Yaskawa INFORM job: OK_R2_O57-69(1)(90,0)_OK_HARDOX.JBI

/JOB
//NAME OK_R2_O57-69(1)(90,0)_OK_HARDOX
///FOLDERNAME X4
//POS
///NPOS 554,554,554,23,0,0
///TOOL 0
///POSTYPE PULSE
///PULSE
C00000=-107863,126513,61876,4074,92941,-4149
C00001=-107635,120046,52933,4022,95106,-4012
C00002=-107385,124787,62548,3925,91623,-4047
C00003=-107289,126429,66937,3891,89767,-4074
C00004=-107289,125685,67059,3890,89310,-4088
C00005=-107289,126429,66937,3891,89767,-4074
C00006=-107447,131976,74605,3936,87910,-4183
C00007=-107368,129085,70604,3913,88881,-4126
C00008=-107503,121805,59343,3962,92067,-4069
C00009=-107756,117289,50059,4061,95463,-4036
C00010=-108153,112100,52912,9904,92668,-10418
C00011=-107537,116907,62411,9707,89272,-10490
C00012=-107296,118643,67053,9639,87306,-10566
C00013=-107296,118210,67408,9641,86871,-10599
C00014=-107296,118643,67053,9639,87306,-10566
C00015=-106873,123308,73383,9530,85780,-10546
C00016=-107051,120523,69599,9574,86686,-10534
C00017=-107734,114067,59645,9761,89532,-10533
C00018=-108357,109439,50420,9963,92855,-10467
C00019=-111395,93808,29792,10909,97789,-10982
C00020=-122185,34205,35653,27729,49230,-19016
C00021=-120981,41909,45488,27980,46968,-19127
C00022=-117396,66636,64308,14609,59928,-14205
C00023=-117396,67398,66227,14722,59162,-14310
C00024=-117396,66924,65038,14651,59635,-14244
C00025=-117026,69424,68003,14605,59045,-14176
C00026=-117396,66924,65038,14651,59635,-14244
C00027=-121567,39659,44448,28509,46708,-19512
C00028=-122801,32028,34766,28268,48928,-19417
C00029=-122836,-30084,-33960,23424,71784,-41222
C00030=-108542,-18181,-29050,8736,76414,-35911
C00031=-108679,-18112,-25517,8852,74315,-36109
C00032=-108679,-17878,-23614,8896,73277,-36184
C00033=-108679,-18015,-24674,8871,73853,-36141
C00034=-101227,-12151,-22997,-5627,79968,-34149
C00035=-100809,-11793,-21323,-5732,79157,-33969
C00036=-99890,-11248,-20900,-5932,79243,-33658
C00037=-100809,-11793,-21323,-5732,79157,-33969
C00038=-119599,-28607,-38623,18108,79564,-38965
C00039=-143809,-13353,-27562,-4151,73883,-14363
C00040=-142866,3813,-3489,-4615,67955,-13814
C00041=-142866,4258,-993,-4658,66653,-13764
C00042=-142866,4067,-2013,-4640,67181,-13786
C00043=-143013,7668,1106,-4588,67106,-13835
C00044=-142866,4067,-2013,-4640,67181,-13786
C00045=-131729,19399,12333,-22118,77640,8494
C00046=-132684,19784,12695,-21959,77361,8191
C00047=-131729,18326,5882,-21907,80820,7904
C00048=-118180,-25123,-37779,-23861,88752,11312
C00049=-84402,-63677,-67114,-22586,99939,48241
C00050=-125926,-77250,-66316,-21080,81833,36437
C00051=-126284,-594,-20029,-15604,88354,35723
C00052=-126284,-509,-12976,-15645,84209,36248
C00053=-124802,3877,-7879,-15893,83645,36839
C00054=-124802,4020,-6552,-15911,82926,36931
C00055=-124802,3943,-7243,-15902,83298,36884
C00056=-123270,3785,-7378,-16131,83600,37383
C00057=-123399,3884,-6575,-16123,83149,37397
C00058=-123813,3922,-6544,-16060,83068,37263
C00059=-123399,3797,-7355,-16113,83568,37342
C00060=-129363,-46213,-49135,-15183,82438,35396
C00061=-131818,-93939,-91511,-4308,83147,7603
C00062=-129147,-104974,-80844,32439,31226,-48978
C00063=-125584,-72667,-62488,33742,33102,-67368
C00064=-122739,-67050,-57509,31022,31859,-65945
C00065=-121864,-64027,-53896,30654,30960,-65755
C00066=-121864,-63651,-52586,31182,30432,-66030
C00067=-121864,-64027,-53896,30654,30960,-65755
C00068=-121821,-59098,-51320,29827,31769,-65322
C00069=-121798,-56590,-49965,29444,32160,-65121
C00070=-121821,-59098,-51320,29827,31769,-65322
C00071=-130221,-55648,-47387,49393,39382,-72629
C00072=-128533,-55969,-47565,48393,38431,-72058
C00073=-122326,-63724,-54491,30711,31580,-65784
C00074=-123406,-65952,-56523,31749,32071,-66325
C00075=-126254,-71501,-61496,34397,33361,-67713
C00076=-120687,-90156,-48971,65843,10407,33929
C00077=-163424,-29173,-12092,69684,68620,47205
C00078=-167450,-15662,-2475,69350,71709,47134
C00079=-157670,-380,9649,68931,65290,48661
C00080=-176833,-62202,-56111,67907,81183,43629
C00081=-171503,-69579,-59831,67744,77015,43718
C00082=-167720,-72113,-59544,67781,73885,43604
C00083=-167720,-71727,-58313,67922,73661,43360
C00084=-167720,-72113,-59544,67781,73885,43604
C00085=-166558,-71597,-59299,67661,73156,43817
C00086=-165333,-70928,-58979,67520,72398,44056
C00087=-166558,-71597,-59299,67661,73156,43817
C00088=-171811,-70314,-60189,67797,77159,43607
C00089=-177694,-60868,-55413,67941,81861,43620
C00090=-178740,-64487,-57291,68086,82281,43176
C00091=-194893,-69888,-59984,68507,92693,40544
C00092=-214988,-85940,-67216,66402,104593,36100
C00093=-106040,-96827,-71490,56175,31560,53564
C00094=-84767,-92802,-92316,-2687,45777,78237
C00095=-91047,27807,-31300,-12206,82587,77963
C00096=-102219,10733,-36282,-6756,75834,75159
C00097=-102220,10108,-35615,-6792,75115,75199
C00098=-102220,9478,-34889,-6816,74349,75240
C00099=-102220,9734,-35191,-6806,74664,75222
C00100=-100300,10893,-34158,-7793,74779,75816
C00101=-100300,10587,-33794,-7807,74401,75842
C00102=-101147,10060,-34263,-7371,74347,75579
C00103=-101076,10802,-35034,-7381,75201,75550
C00104=-95480,80551,28809,-25074,106745,88551
C00105=-95760,77540,27472,-24942,106007,88613
C00106=-95760,76990,28122,-24849,105386,88749
C00107=-95760,77103,27982,-24868,105516,88720
C00108=-96959,80585,32244,-24647,104424,88528
C00109=-96959,80447,32426,-24624,104257,88565
C00110=-96409,78816,30426,-24722,104765,88651
C00111=-100062,100483,54273,-17494,109954,86476
C00112=-106835,71636,17530,-18824,115982,83026
C00113=-106612,70519,18025,-18669,115194,83244
C00114=-106612,70167,18360,-18604,114826,83306
C00115=-106612,70294,18237,-18628,114960,83283
C00116=-107711,74369,23131,-18489,113861,83072
C00117=-107711,74237,23265,-18465,113717,83098
C00118=-107290,72601,21292,-18521,114156,83175
C00119=-107383,75666,22241,-18686,115079,82983
C00120=-103109,12889,-33455,-26802,75758,89629
C00121=-108969,18301,-24187,-24197,71491,88552
C00122=-108969,17786,-23402,-24296,70807,88698
C00123=-108969,17914,-23607,-24271,70984,88661
C00124=-107778,14157,-27071,-24854,71490,88973
C00125=-107778,13979,-26794,-24889,71252,89025
C00126=-108147,15245,-25637,-24709,71092,88927
C00127=-108126,15683,-27040,-24578,72092,88718
C00128=-100567,37939,-6230,-27391,72804,90359
C00129=-100865,37186,-5596,-27353,72020,90442
C00130=-100865,36842,-5001,-27431,71534,90560
C00131=-100865,36955,-5200,-27406,71694,90520
C00132=-99747,33295,-8939,-27886,72410,90754
C00133=-99747,33126,-8648,-27924,72173,90813
C00134=-100160,34398,-7357,-27744,71921,90725
C00135=-100129,35026,-9173,-27563,73215,90418
C00136=-110911,33745,-10798,1686,65996,79969
C00137=-110596,33512,-9684,1507,65185,80063
C00138=-110596,33168,-9124,1512,64663,80058
C00139=-110596,33307,-9355,1509,64876,80061
C00140=-109674,30137,-12540,942,65194,80377
C00141=-109674,29950,-12234,942,64908,80377
C00142=-110141,31373,-10814,1228,64772,80217
C00143=-110010,31979,-12214,1138,65943,80273
C00144=-98269,67962,25517,-6197,61564,84446
C00145=-97899,69655,29924,-6541,59762,84684
C00146=-97899,69423,30622,-6575,59215,84716
C00147=-97899,69536,30274,-6557,59484,84700
C00148=-96720,65812,25908,-7249,60348,85083
C00149=-96720,65654,26340,-7274,60006,85106
C00150=-97107,66951,27854,-7050,59711,84981
C00151=-96963,66930,26864,-7100,60316,84996
C00152=-95444,-1255,-51083,-7343,73273,84703
C00153=-87441,-44243,-81586,-12090,70841,87391
C00154=-204042,-120915,-85873,62426,87530,23210
C00155=-200540,-66438,-67217,63628,100285,-15829
C00156=-127293,-88890,-117674,21964,112183,-47373
C00157=-127884,-113870,-117586,20406,100261,-49782
C00158=-126455,-94233,-83658,19548,96625,-49926
C00159=-122769,-95152,-80887,19686,93685,-49072
C00160=-121257,-92855,-76623,19731,91957,-48808
C00161=-121256,-92184,-75240,19721,91480,-48885
C00162=-121257,-92855,-76623,19731,91957,-48808
C00163=-119709,-92847,-76620,19813,91585,-48312
C00164=-118447,-92805,-76604,19874,91287,-47906
C00165=-121134,-93057,-78029,19757,92646,-48652
C00166=-122616,-92853,-79205,19699,93786,-49000
C00167=-126246,-91944,-81970,19569,96706,-49837
C00168=-116739,-91029,-87152,-11175,94833,69838
C00169=-118638,-93558,-84500,-11112,91693,69464
C00170=-121559,-94813,-81066,-11067,88585,68734
C00171=-121559,-94454,-79960,-11067,88097,68778
C00172=-121559,-94813,-81066,-11067,88585,68734
C00173=-121580,-97932,-82261,-11067,87731,68801
C00174=-121559,-94813,-81066,-11067,88585,68734
C00175=-124478,-94674,-81011,-11026,88221,67759
C00176=-121559,-94813,-81066,-11067,88585,68734
C00177=-121199,-93273,-83309,-11082,90766,68663
C00178=-119237,-90980,-86060,-11143,93854,69064
C00179=-119262,-91078,-98551,-11400,101347,68370
C00180=-119262,-88450,-105465,-11733,106843,67839
C00181=-123634,-129086,-124562,18007,62786,-21453
C00182=-124713,-112307,-109989,18584,62695,-21889
C00183=-121750,-102661,-104576,16897,63614,-20597
C00184=-120661,-96847,-100545,16291,63882,-20142
C00185=-120661,-96945,-99213,16408,63045,-20264
C00186=-120661,-96847,-100545,16291,63882,-20142
C00187=-119434,-96825,-100537,15680,63651,-19709
C00188=-118199,-96764,-100511,15059,63439,-19270
C00189=-119434,-96825,-100537,15680,63651,-19709
C00190=-120468,-95018,-99831,16130,64325,-20004
C00191=-120473,-92385,-98782,16042,65005,-19908
C00192=-120468,-95018,-99831,16130,64325,-20004
C00193=-121400,-102567,-103315,16828,62845,-20579
C00194=-124338,-112119,-108698,18515,61948,-21869
C00195=-115152,-110094,-108973,-21966,66789,27187
C00196=-118701,-101887,-103909,-20282,66922,25804
C00197=-120033,-96498,-99821,-19662,66842,25314
C00198=-120033,-96571,-98630,-19770,66116,25442
C00199=-120033,-96498,-99821,-19662,66842,25314
C00200=-121038,-96503,-99823,-19217,66607,24975
C00201=-122863,-96447,-99800,-18396,66209,24352
C00202=-121038,-96503,-99823,-19217,66607,24975
C00203=-121031,-93073,-98698,-19079,67622,24806
C00204=-121028,-91162,-97925,-19016,68103,24728
C00205=-121031,-93073,-98698,-19079,67622,24806
C00206=-119849,-101075,-102503,-19842,66224,25492
C00207=-116381,-109262,-107580,-21511,66068,26853
C00208=-114174,-113759,-109466,-25218,61256,29915
C00209=-117999,-105066,-104585,-23039,61495,28291
C00210=-119436,-99712,-100384,-22286,61259,27759
C00211=-119436,-99710,-99356,-22420,60673,27881
C00212=-119436,-99712,-100384,-22286,61259,27759
C00213=-121229,-99730,-100389,-21374,60785,27131
C00214=-123455,-99637,-100354,-20211,60254,26337
C00215=-121229,-99730,-100389,-21374,60785,27131
C00216=-121193,-87849,-97584,-20616,64895,26352
C00217=-121184,-85182,-96456,-20515,65531,26236
C00218=-121193,-87849,-97584,-20616,64895,26352
C00219=-119818,-94456,-100985,-21520,64018,27049
C00220=-116346,-102514,-105912,-23431,63914,28430
C00221=-120616,-96535,-104175,-23887,64719,45568
C00222=-120616,-96992,-102054,-24182,63306,45881
C00223=-136549,-91664,-102215,-2850,64532,40154
C00224=-118869,-97062,-101163,-25162,63282,46587
C00225=-120614,-98220,-102778,-24220,63138,45920
C00226=-133771,-94843,-111628,-11760,91195,37379
C00227=-135495,-95953,-105009,-10406,87462,38794
C00228=-135817,-95923,-103691,-10152,86855,39072
C00229=-120616,-96793,-103087,-23408,87451,42960
C00230=-120617,-96070,-105685,-23410,89266,42604
C00231=-120635,-118119,-124325,-17957,114364,37370
C00232=-107148,-122068,-106720,-37591,45003,56343
C00233=-107143,-118125,-97071,-40168,41922,57944
C00234=-107140,-117153,-94914,-40772,41285,58308
C00235=-108761,-111076,-92035,-38763,41593,57087
C00236=-105115,-116142,-93852,-42098,42144,59139
C00237=-107012,-118507,-95796,-40965,41228,58425
C00238=-106625,-124982,-112623,-27698,77800,49761
C00239=-108670,-124346,-112001,-25564,83023,48254
C00240=-122914,-112386,-108022,-9565,118901,48106
C00241=-107149,-124464,-114807,-14035,115464,42498
C00242=-107153,-124980,-118069,-14274,117155,42276
C00243=-120683,-72727,-118704,-1403,106780,1205
C00244=-120616,-97084,-101761,23685,56760,-46645
C00245=-120615,-97341,-97713,24403,54354,-47226
C00246=-120615,-97245,-95574,24781,53197,-47519
C00247=-113473,-96585,-93861,15515,48754,-41599
C00248=-120613,-98403,-96349,24817,53089,-47545
C00249=-122362,-97151,-94697,25998,53280,-48291
C00250=-118726,-95773,-106258,22948,89010,-41713
C00251=-118527,-107245,-109313,22939,85243,-42364
C00252=-120617,-95328,-107797,23350,90604,-42068
C00253=-120618,-93989,-110172,23402,92584,-41681
C00254=-120619,-87370,-116055,23793,99045,-40394
C00255=-120619,-87370,-116055,23793,99045,-40394
C00256=-120618,-86394,-114990,-8935,74593,-77376
C00257=-120618,-89943,-112390,-9089,71210,-77123
C00258=-120618,-91094,-111253,-9157,69935,-77026
C00259=-120921,-87010,-110025,-8929,71231,-77225
C00260=-120616,-91696,-112687,-9127,70502,-77069
C00261=-120617,-91433,-110915,-9280,69085,-76949
C00262=-120617,-91707,-110620,-9342,68290,-76888
C00263=-120617,-92092,-110153,-9289,66860,-76810
C00264=-120617,-92703,-109346,-8604,64312,-76688
C00265=-120617,-93084,-108807,-7222,62458,-76641
C00266=-120617,-93193,-108666,-5837,61715,-76664
C00267=-120618,-90875,-111661,-5103,64613,-76670
C00268=-120618,-90809,-111742,-4197,64653,-76687
C00269=-120618,-90545,-112027,-2634,65244,-76730
C00270=-120618,-90001,-112556,-1051,66686,-76779
C00271=-120618,-89211,-113241,130,68806,-76818
C00272=-120618,-88484,-113805,667,70701,-76840
C00273=-120618,-87123,-114601,725,72803,-76709
C00274=-120619,-86169,-115177,666,75079,-76754
C00275=-120619,-85009,-115798,-44,77805,-76866
C00276=-120619,-84186,-116189,-1368,79788,-77043
C00277=-120619,-83945,-116287,-2643,80551,-77203
C00278=-118270,-87908,-113898,-4548,77310,-76315
C00279=-117006,-87882,-113777,-5977,77383,-75992
C00280=-115001,-87936,-113393,-8376,77055,-75464
C00281=-113157,-88199,-112730,-10795,75966,-74930
C00282=-112003,-88721,-111920,-12625,74164,-74513
C00283=-111959,-89151,-111512,-13141,72976,-74431
C00284=-114352,-90005,-111461,-12180,71784,-75105
C00285=-117604,-90791,-111341,-10710,70486,-76060
C00286=-117404,-89600,-112462,-10735,71791,-76111
C00287=-116906,-85938,-115017,-10812,75246,-76259
C00288=-120614,-97623,-100799,-20300,88883,51757
C00289=-120614,-96302,-87355,-20440,81742,52958
C00290=-120613,-95405,-83784,-20521,80111,53236
C00291=-127344,-108772,-84900,-17713,65232,40253
C00292=-119108,-93712,-82042,-20736,80300,53753
C00293=-120703,-96440,-84059,-20528,79748,53266
C00294=-121654,-94959,-82200,-16195,85067,56749
C00295=-121447,-94482,-79045,-16244,83477,57034
C00296=-120534,-97306,-80078,-13287,88870,68293
C00297=-120613,-95181,-82964,-13310,91650,67966
C00298=-120614,-96223,-86939,-13345,93512,67766
C00299=-120615,-97634,-95801,-13498,98116,67263
C00300=-121294,-114205,-91205,24827,58618,-34956
C00301=-120612,-94063,-79189,30374,49118,-27390
C00302=-120612,-92317,-74276,31337,47279,-28045
C00303=-120611,-91635,-72532,31685,46659,-28276
C00304=-117825,-85297,-69483,27706,45876,-25590
C00305=-120609,-92794,-73597,31655,46709,-28256
C00306=-122365,-91337,-71823,32796,47086,-29053
C00307=-115287,-110447,-90354,20374,67075,-37718
C00308=-116232,-100454,-77072,21254,66209,-40580
C00309=-116013,-94136,-76050,20295,81458,-56297
C00310=-120612,-93792,-78416,23522,88402,-60481
C00311=-120613,-94966,-82014,23532,89885,-60189
C00312=-192979,-49879,-84133,31949,90821,-59300
C00313=-226136,-49296,-77583,43048,96139,-60221
C00314=-194231,-43574,-37464,64429,96533,35524
C00315=-168190,-921,2356,69742,86936,65420
C00316=-167171,-9679,-4727,69794,80481,66551
C00317=-161668,-12899,-4972,71887,72051,48991
C00318=-157343,-12771,-6150,68681,68498,39910
C00319=-156881,-17849,-10944,69825,79076,66625
C00320=-156054,-17027,-11609,69675,78824,67093
C00321=-157320,-12846,-6207,68680,68481,39912
C00322=-155303,-14498,-7398,68413,65801,40416
C00323=-150761,-18705,-10675,67104,57790,42164
C00324=-154138,4950,8277,69166,76187,38481
C00325=-154445,-11009,-7055,66235,75211,55885
C00326=-154064,-10379,-10377,61252,81435,65690
C00327=-159305,-13086,-7363,68622,70046,39902
C00328=-160610,-11568,-6196,68690,70948,39749
C00329=-179726,-19719,-12316,69264,83687,37039
C00330=-180202,-65513,-36112,70171,79517,38597
C00331=-171321,-47804,-23743,70196,73038,45095
C00332=-120855,-117042,-83065,287,50429,-281
C00333=-120852,-56541,-79529,233,79340,-219
C00334=-120696,51333,26745,175,69370,-180
C00335=-120686,107911,74673,172,68949,-177
C00336=-120685,95088,60632,169,71000,-174
C00337=-122318,97205,64688,817,69601,-751
C00338=-120685,108202,77433,173,67399,-179
C00339=-120704,104217,73450,180,67803,-185
C00340=-122286,97202,64700,804,69591,-740
C00341=-121454,98107,65862,475,69334,-448
C00342=-120585,97922,65623,2034,69446,-1841
C00343=-122017,99369,67601,7878,69886,-7136
C00344=-124401,105713,75936,15606,71119,-14640
C00345=-128119,115493,91326,26372,70058,-18277
C00346=-128088,115464,91288,26362,70055,-18265
C00347=-119886,111402,95174,38234,57086,-30403
C00348=-120666,108818,81293,29360,75518,-26461
C00349=-140740,108253,75800,14319,69459,-12393
C00350=-141155,96820,62941,14306,71509,-12294
C00351=-143909,115216,86261,19079,74712,-18279
C00352=-140740,108512,78347,14450,68068,-12565
C00353=-141173,105757,75971,14609,68190,-12710
C00354=-142377,104065,71962,18453,77277,-17320
C00355=-143915,117471,89727,22794,77825,-23537
C00356=-139477,109798,84410,35996,86879,-36501
C00357=-140751,108928,81956,36051,87607,-36108
C00358=-140752,108346,78971,36051,88864,-35697
C00359=-147823,62894,38016,27898,90947,-27507
C00360=-160213,20954,5847,52912,104038,-48859
C00361=-159152,20729,17995,59071,100827,-50067
C00362=-155802,40777,37843,59069,97737,-50212
C00363=-160195,38796,31307,59203,102054,-49818
C00364=-156773,55935,3033,15469,106475,-467
C00365=-153918,39963,-12238,-14336,97152,19223
C00366=-159942,42906,-84,-7000,88493,12017
C00367=-161832,44450,4966,-4658,85344,9495
C00368=-160451,43537,6688,-5079,83896,9996
C00369=-170176,47751,11203,12092,85800,-8664
C00370=-172574,61876,26837,20283,90605,-20342
C00371=-175474,59660,23243,20803,92313,-21058
C00372=-176824,52719,4578,21456,100048,-20156
C00373=-152577,48148,-11201,-5231,110173,9097
C00374=-182779,-40861,-76585,4205,87735,83212
C00375=-189334,-126614,-108463,44477,62316,64668
C00376=-120096,-126434,-88762,51835,16555,74218
C00377=-139248,-82584,-73342,59042,45862,69599
C00378=-136350,-83647,-73803,58003,43942,70198
C00379=-130421,-76673,-73912,46604,46265,76427
C00380=-135820,-86240,-74234,58721,43036,69743
C00381=-135177,-84196,-74622,57263,43352,70634
C00382=-130462,-76664,-73908,46626,46288,76415
C00383=-118284,-90424,-77484,27464,26422,76602
C00384=-134750,-71454,-68054,46452,38063,58888
C00385=-143711,-58767,-60463,57749,51756,38253
C00386=-120675,-86248,-74914,23863,24288,53303
C00387=-120674,-86256,-74917,23863,24286,53303
C00388=-120096,-126434,-88762,51835,16555,74218
C00389=-118534,-85327,-101542,-31688,82312,3081
C00390=-123235,4833,-40404,-29868,88268,-211
C00391=-160796,40344,30640,-17217,54638,-7315
C00392=-160797,40341,30637,-17217,54638,-7315
C00393=-160797,40341,30637,-17217,54638,-7315
C00394=-160252,39151,28676,-17378,55324,-7200
C00395=-161178,38223,28434,-16963,54814,-7508
C00396=-160796,40350,30646,-17218,54637,-7315
C00397=-160795,40351,30648,-17218,54637,-7314
C00398=-160794,40354,30651,-17218,54637,-7314
C00399=-134054,6396,-12292,-27269,70214,305
C00400=-134055,6392,-12295,-27269,70214,305
C00401=-134055,6392,-12295,-27269,70214,305
C00402=-133335,6117,-13247,-27465,70843,432
C00403=-134208,4264,-14132,-27207,70198,248
C00404=-134055,6400,-12288,-27269,70214,305
C00405=-134054,6402,-12286,-27269,70214,305
C00406=-134054,6405,-12283,-27270,70214,305
C00407=-134054,6378,-12307,-27269,70215,305
C00408=-110297,97127,46558,-158,86609,-5885
C00409=-106536,103923,39499,6534,95353,-6477
C00410=-105914,112602,52325,6316,91893,-6465
C00411=-107411,115180,62232,6738,87264,-7175
C00412=-107307,119116,66280,6709,86790,-7167
C00413=-105927,112591,52310,6320,91897,-6469
C00414=-107439,122836,73336,-765,83341,-3278
C00415=-107821,123137,73841,-645,83181,-3398
C00416=-102914,145277,103073,-11065,82212,10729
C00417=-102506,149279,108574,-13236,82700,14235
C00418=-102941,142782,99507,-15695,87156,18184
C00419=-102438,125149,73506,-15865,93942,17486
C00420=-103348,95167,36366,-12069,90690,17205
C00421=-107306,118463,66661,-801,85196,-3245
C00422=-107311,128667,66498,14067,94509,-10827
C00423=-105409,128969,69208,9127,93984,-11176
C00424=-104752,117595,57274,7632,88999,-11570
C00425=-107310,126688,66629,14039,93443,-10948
C00426=-107566,122823,62593,14116,93966,-10970
C00427=-105955,108102,46748,11418,87672,-11524
C00428=-106075,110081,48628,12407,89224,-11272
C00429=-104774,107445,45071,11972,89867,-10810
C00430=-104167,107349,44943,11766,89817,-10628
C00431=-103614,108174,46048,11576,89495,-10489
C00432=-105019,105279,39955,12261,92654,-10576
C00433=-107312,128730,66586,14067,94488,-10830
C00434=-113054,107191,42951,15619,98894,-12042
C00435=-132655,20555,-34602,20500,105579,-17250
C00436=-120395,-75677,-109491,17431,99945,-14261
C00437=-120179,-75618,-109521,17213,99976,-84333
C00438=-116382,-32242,-70046,11239,66277,-88684
C00439=-117174,1233,-44945,11588,68097,-88765
C00440=-107946,15126,-37900,-11639,87566,-88486
C00441=-109328,12351,-36379,-11088,85080,-88672
C00442=-109363,12887,-35894,-11074,85053,-88680
C00443=-109363,12887,-35894,-11074,85053,-88680
C00444=-111924,52141,-3629,-8112,105606,-90388
C00445=-112776,77755,26238,-11993,114409,-73073
C00446=-113379,76285,24444,-12049,114668,-73314
C00447=-123052,55319,260,-15299,117047,-77561
C00448=-123040,57609,790,-15431,117871,-77674
C00449=-105167,32161,-17434,-30422,80375,-70409
C00450=-107613,28576,-14101,-29706,76191,-70169
C00451=-107575,27990,-14679,-29717,76251,-70170
C00452=-107056,35688,-9010,-30442,81556,-71715
C00453=-107174,35007,-9708,-30392,81586,-71765
C00454=-107604,33855,-10883,-30216,81557,-71912
C00455=-106755,42437,-3209,-32490,86542,-73631
C00456=-116032,20896,-23074,-32399,83882,-77024
C00457=-116007,21026,-25434,-32353,85183,-77388
C00458=-117682,52698,-4766,-11690,95851,-49632
C00459=-117257,51519,-1008,-11752,93047,-49237
C00460=-117197,51091,-1482,-11772,93125,-49226
C00461=-117014,50506,-2129,-11828,93245,-49180
C00462=-116272,43957,-7629,-12215,89681,-48654
C00463=-116775,24502,-20794,-9432,75702,-46765
C00464=-100350,61255,17965,-17507,73385,-41100
C00465=-98698,68325,24845,-19999,74224,-56366
C00466=-96693,71424,29264,-24904,74423,-56480
C00467=-96693,72048,27992,-24790,75430,-56697
C00468=-111009,19081,-28851,-17902,79273,-62219
C00469=-101550,-89760,-106531,-22768,73782,-58094
C00470=-120731,-81008,-115648,-105,86416,-81801
C00471=-120675,-24654,-47163,-132,73228,-81771
C00472=-120676,-24640,-47153,-131,73229,-81771
C00473=-121102,-22780,-44290,48,72423,-81914
C00474=-120676,-24370,-48215,-131,74021,-81772
C00475=-121750,-24626,-47144,317,73232,-82133
C00476=-121088,-18910,-41523,41,72708,-81911
C00477=-120676,-24640,-47153,-131,73229,-81771
C00478=-120672,-32524,-49889,-133,70864,-81769
C00479=-86683,-40445,-63075,-13763,77736,-70672
C00480=-103499,26970,-9106,-7161,77072,-76192
C00481=-140778,108078,66600,-20509,92089,-48724
C00482=-140778,108101,66629,-20508,92083,-48723
C00483=-140777,108123,66659,-20508,92077,-48722
C00484=-140791,110557,71328,-20474,90549,-48468
C00485=-140777,108420,65802,-20527,92715,-48830
C00486=-141368,109052,67884,-20414,91674,-48860
C00487=-140538,117676,80864,-20492,88534,-48038
C00488=-140777,108123,66659,-20508,92077,-48722
C00489=-140778,108101,66629,-20508,92083,-48723
C00490=-140778,108101,66629,-20508,92083,-48723
C00491=-140778,108122,66658,-20508,92077,-48722
C00492=-140768,108703,68758,-20489,91145,-48562
C00493=-140777,108420,65801,-20527,92715,-48830
C00494=-141368,109051,67883,-20414,91674,-48860
C00495=-140511,115176,77354,-20500,89363,-48171
C00496=-140778,108122,66658,-20508,92077,-48722
C00497=-140778,108100,66628,-20508,92083,-48723
C00498=-140778,108078,66599,-20509,92089,-48724
C00499=-126581,14025,-47477,-25241,115824,-48542
C00500=-159492,92702,46653,-29136,105568,-44545
C00501=-162149,88036,41181,-28914,105145,-45798
C00502=-163325,88052,47564,-28312,101300,-45262
C00503=-160866,111719,71725,-28335,100123,-43674
C00504=-160864,108336,66000,-28535,101703,-44070
C00505=-164354,88224,47874,-28236,100875,-45547
C00506=-160866,108108,66623,-28476,101259,-43959
C00507=-161429,110004,69125,-28389,100573,-44000
C00508=-160867,107600,68720,-43807,97992,-44930
C00509=-160869,107245,72152,-43546,96305,-44200
C00510=-160853,112270,81548,-43267,93953,-43186
C00511=-160872,111361,79145,-43345,94689,-43509
C00512=-160869,107230,72446,-43527,96165,-44140
C00513=-161852,112523,81931,-43214,93388,-43402
C00514=-160870,107231,72133,-43547,96307,-44201
C00515=-160868,107586,68702,-43807,97995,-44932
C00516=-160873,107541,68625,-43810,98010,-44941
C00517=-160875,107181,72050,-43549,96324,-44211
C00518=-160969,112164,81513,-43259,93871,-43205
C00519=-160878,111286,79028,-43348,94711,-43521
C00520=-160875,107165,72344,-43530,96184,-44151
C00521=-161946,112277,81723,-43208,93342,-43426
C00522=-160876,107167,72031,-43549,96326,-44212
C00523=-160874,107528,68607,-43810,98012,-44942
C00524=-160865,108116,66633,-19225,80466,79641
C00525=-160864,108012,67019,-19239,80191,79685
C00526=-160902,111102,73963,-19378,77641,80084
C00527=-160868,111461,73140,-19346,78303,79987
C00528=-160865,107941,67240,-19247,80028,79711
C00529=-161896,111383,74336,-19093,77331,79779
C00530=-160866,107998,67001,-19238,80195,79684
C00531=-160866,108102,66615,-19224,80470,79640
C00532=-141960,25007,-13534,-18907,77065,75548
C00533=-148396,38776,-224,-4331,80270,75408
C00534=-147937,42862,4060,-4507,79758,75574
C00535=-147586,38479,-2882,-4613,81790,75612
C00536=-132676,28155,-16568,-22865,92034,69453
C00537=-139622,-24488,-52979,-20482,85647,66084
C00538=-105595,-117820,-100492,-25848,75539,72989
C00539=-106580,-108863,-97500,-25415,77736,72126
C00540=-109054,-118504,-91401,-16987,64899,66879
C00541=-114351,-116427,-87550,-15194,62531,65147
C00542=-119485,-94955,-76898,-12502,65960,62737
C00543=-99170,-109633,-81201,-29999,68590,70531
C00544=-97263,-108225,-79726,-30318,69111,71170
C00545=-119688,-71486,-66798,-11989,71648,62069
C00546=-119489,-72073,-70371,-11931,73536,61952
C00547=-119715,-43131,-54580,-11630,78554,61387
C00548=-119934,-43288,-51446,-11646,76556,61502
C00549=-120006,-17553,-34071,-11532,79027,61243
C00550=-119832,-16968,-37707,-11506,81540,61066
C00551=-138269,-21321,-44343,15851,46320,74175
C00552=-176671,-154466,-104215,64912,39697,45563
C00553=-34524,-124554,-102946,40349,70974,61921
BC00000=290556,778984,53
BC00001=296477,827832,53
BC00002=296477,827832,53
BC00003=296477,827832,52
BC00004=296477,827832,52
BC00005=296477,827832,52
BC00006=296477,827832,52
BC00007=296477,827832,52
BC00008=296477,827832,53
BC00009=296477,827832,53
BC00010=305680,824697,66927
BC00011=305680,824697,66927
BC00012=305680,824697,66927
BC00013=305680,824697,66927
BC00014=305680,824697,66927
BC00015=305680,824697,66927
BC00016=305680,824697,66927
BC00017=305680,824697,66927
BC00018=305680,824697,66927
BC00019=305680,824697,66927
BC00020=269068,808420,256770
BC00021=269068,808420,256770
BC00022=269068,808420,256770
BC00023=269068,808420,256770
BC00024=269068,808420,256770
BC00025=269068,808420,256770
BC00026=269068,808420,256770
BC00027=269068,808420,256770
BC00028=269068,808420,256770
BC00029=269068,808420,256770
BC00030=269068,808420,256770
BC00031=269068,808420,256770
BC00032=269068,808420,256770
BC00033=269068,808420,256770
BC00034=269068,808420,256770
BC00035=269068,808420,256770
BC00036=269068,808420,256770
BC00037=269068,808420,256770
BC00038=269068,808420,256770
BC00039=269068,808420,256770
BC00040=269068,808420,256770
BC00041=269068,808420,256770
BC00042=269068,808420,256770
BC00043=269068,808420,256770
BC00044=269068,808420,256770
BC00045=269068,808420,256770
BC00046=269068,808420,256770
BC00047=269068,808420,256770
BC00048=269068,808420,256770
BC00049=269068,722620,256770
BC00050=178494,722620,256770
BC00051=178494,722620,256770
BC00052=178494,722620,256770
BC00053=178494,722620,256770
BC00054=178494,722620,256770
BC00055=178494,722620,256770
BC00056=178494,722620,256770
BC00057=178494,722620,256770
BC00058=178494,722620,256770
BC00059=178494,722620,256770
BC00060=178494,722620,256770
BC00061=138756,709064,202273
BC00062=61964,682869,96959
BC00063=15,683519,90542
BC00064=15,683519,90542
BC00065=15,683519,90542
BC00066=15,683519,90542
BC00067=15,683519,90542
BC00068=15,683519,90542
BC00069=15,683519,90542
BC00070=15,683519,90542
BC00071=15,683519,90542
BC00072=15,683519,90542
BC00073=15,683519,90542
BC00074=15,683519,90542
BC00075=15,683519,90542
BC00076=1273,683756,232707
BC00077=15,671225,229408
BC00078=15,671225,229408
BC00079=16,671226,229406
BC00080=15,740766,97992
BC00081=15,744979,78990
BC00082=15,746665,71384
BC00083=15,746665,71384
BC00084=15,746665,71384
BC00085=15,746665,71384
BC00086=15,746665,71384
BC00087=15,746665,71384
BC00088=15,744091,71514
BC00089=15,739878,90515
BC00090=15,739878,90515
BC00091=15,739878,90515
BC00092=15,739878,90515
BC00093=15,678682,90515
BC00094=86538,678682,90515
BC00095=86538,751250,55
BC00096=86538,751250,55
BC00097=86537,751250,51
BC00098=86537,751250,51
BC00099=86537,751250,51
BC00100=86537,751250,51
BC00101=86537,751250,51
BC00102=86537,751250,51
BC00103=86537,751250,51
BC00104=86537,751250,51
BC00105=86537,751250,51
BC00106=86537,751250,51
BC00107=86537,751250,51
BC00108=86537,751250,51
BC00109=86537,751250,51
BC00110=86537,751250,51
BC00111=86537,751250,51
BC00112=86537,751250,51
BC00113=86537,751250,51
BC00114=86537,751250,51
BC00115=86537,751250,51
BC00116=86537,751250,51
BC00117=86537,751250,51
BC00118=86537,751250,51
BC00119=86537,751250,51
BC00120=86537,751250,51
BC00121=86537,751250,51
BC00122=86537,751250,51
BC00123=86537,751250,51
BC00124=86537,751250,51
BC00125=86537,751250,51
BC00126=86537,751250,51
BC00127=86537,751250,51
BC00128=86537,751250,51
BC00129=86537,751250,51
BC00130=86537,751250,51
BC00131=86537,751250,51
BC00132=86537,751250,51
BC00133=86537,751250,51
BC00134=86537,751250,51
BC00135=86537,751250,51
BC00136=86537,751250,51
BC00137=86537,751250,51
BC00138=86537,751250,51
BC00139=86537,751250,51
BC00140=86537,751250,51
BC00141=86537,751250,51
BC00142=86537,751250,51
BC00143=86537,751250,51
BC00144=86537,751250,51
BC00145=86537,751250,51
BC00146=86537,751250,51
BC00147=86537,751250,51
BC00148=86537,751250,51
BC00149=86537,751250,51
BC00150=86537,751250,51
BC00151=86537,751250,51
BC00152=86537,751250,51
BC00153=86537,663623,51
BC00154=4537,733723,217212
BC00155=80822,696048,563603
BC00156=35157,680076,1075175
BC00157=35157,770360,1075175
BC00158=34361,771324,1075175
BC00159=34361,771324,1075175
BC00160=34361,771324,1075175
BC00161=34361,771324,1075175
BC00162=34361,771324,1075175
BC00163=34361,771324,1075175
BC00164=34361,771324,1075175
BC00165=34361,771324,1075175
BC00166=34361,771324,1075175
BC00167=34361,771324,1075175
BC00168=42797,766692,1075175
BC00169=42797,766692,1075175
BC00170=42797,766692,1075175
BC00171=42797,766692,1075175
BC00172=42797,766692,1075175
BC00173=42797,766692,1075175
BC00174=42797,766692,1075175
BC00175=42797,766692,1075175
BC00176=42797,766692,1075175
BC00177=42797,766692,1075175
BC00178=42797,766692,1075175
BC00179=42797,766692,1075175
BC00180=42797,766692,1075175
BC00181=146022,859779,1075175
BC00182=146022,859779,1075175
BC00183=146022,859779,1075175
BC00184=146022,859779,1075175
BC00185=146022,859779,1075175
BC00186=146022,859779,1075175
BC00187=146022,859779,1075175
BC00188=146022,859779,1075175
BC00189=146022,859779,1075175
BC00190=146022,859779,1075175
BC00191=146022,859779,1075175
BC00192=146022,859779,1075175
BC00193=146022,859779,1075175
BC00194=146022,859779,1075175
BC00195=176049,857561,1075175
BC00196=176049,857561,1075175
BC00197=176049,857561,1075175
BC00198=176049,857561,1075175
BC00199=176049,857561,1075175
BC00200=176049,857561,1075175
BC00201=176049,857561,1075175
BC00202=176049,857561,1075175
BC00203=176049,857561,1075175
BC00204=176049,857561,1075175
BC00205=176049,857561,1075175
BC00206=176049,857561,1075175
BC00207=176049,857561,1075175
BC00208=129734,841826,1075175
BC00209=129734,841826,1075175
BC00210=129734,841826,1075175
BC00211=129734,841826,1075175
BC00212=129734,841826,1075175
BC00213=129734,841826,1075175
BC00214=129734,841826,1075175
BC00215=129734,841826,1075175
BC00216=129734,841826,1075175
BC00217=129734,841826,1075175
BC00218=129734,841826,1075175
BC00219=129734,841826,1075175
BC00220=129734,841826,1075175
BC00221=142153,845657,1075175
BC00222=136701,849303,1075175
BC00223=134520,850762,1075175
BC00224=134520,850762,1075175
BC00225=134520,850762,1075175
BC00226=137516,886222,1075172
BC00227=137720,849041,1075174
BC00228=137762,841415,1075175
BC00229=140007,840932,1075175
BC00230=145619,839727,1075175
BC00231=180456,929432,1075175
BC00232=168021,846183,1075175
BC00233=168042,846186,1075175
BC00234=163006,851102,1075175
BC00235=160992,853068,1075175
BC00236=160992,853068,1075175
BC00237=160992,853068,1075175
BC00238=169557,896858,1075175
BC00239=171239,895275,1075172
BC00240=158426,945505,1075171
BC00241=160107,947347,1075175
BC00242=164973,949360,1075175
BC00243=157894,860706,1075175
BC00244=127221,848277,1075175
BC00245=127232,848278,1075175
BC00246=132508,852516,1075175
BC00247=134618,854212,1075171
BC00248=134619,854211,1075175
BC00249=134619,854211,1075175
BC00250=128708,899486,1075175
BC00251=128708,899486,1075175
BC00252=126448,894646,1075175
BC00253=120840,893399,1075175
BC00254=120819,893396,1075175
BC00255=108659,806260,1075175
BC00256=397033,866889,1075175
BC00257=396343,869401,1075175
BC00258=396067,870405,1075175
BC00259=396067,870405,1075175
BC00260=396067,870405,1075175
BC00261=391503,868887,1075175
BC00262=388851,867701,1075175
BC00263=387842,866199,1075175
BC00264=385581,863689,1075175
BC00265=382314,862051,1075175
BC00266=379450,861705,1075175
BC00267=374365,881250,1075175
BC00268=372628,881564,1075175
BC00269=369853,882526,1075175
BC00270=367245,884287,1075175
BC00271=365527,886651,1075175
BC00272=365120,888691,1075175
BC00273=386897,893714,1075175
BC00274=387767,895993,1075175
BC00275=389889,898568,1075175
BC00276=393093,900280,1075175
BC00277=395952,900656,1075175
BC00278=398174,881178,1075175
BC00279=398174,880854,1075175
BC00280=398174,879840,1075175
BC00281=398174,877989,1075175
BC00282=398174,875535,1075175
BC00283=398174,874097,1075175
BC00284=398174,872876,1075175
BC00285=398174,871457,1075175
BC00286=398174,870453,1075175
BC00287=398174,867941,1075175
BC00288=52330,766929,1075175
BC00289=52330,766929,1075175
BC00290=47260,766939,1075175
BC00291=45232,766943,1075175
BC00292=45232,766943,1075175
BC00293=45232,766943,1075175
BC00294=39669,775379,1075175
BC00295=48611,761121,1075175
BC00296=43094,771298,1075175
BC00297=44336,772357,1075175
BC00298=47441,775005,1075175
BC00299=47420,775002,1075175
BC00300=32781,783617,1075175
BC00301=26171,746916,1075175
BC00302=26181,746918,1075175
BC00303=30773,752599,1075175
BC00304=32609,754871,1075175
BC00305=32609,754871,1075175
BC00306=32609,754871,1075175
BC00307=29513,796201,1075175
BC00308=29656,745498,1075175
BC00309=30736,758476,1075175
BC00310=29625,769411,1075175
BC00311=24737,771387,1075175
BC00312=181441,722385,1075175
BC00313=206367,695978,993979
BC00314=43511,699656,343050
BC00315=15,700638,169199
BC00316=15,700493,176682
BC00317=15,702608,172046
BC00318=15,703868,169284
BC00319=15,702762,156281
BC00320=15,702762,156281
BC00321=15,703868,169284
BC00322=15,698813,169275
BC00323=15,689550,169221
BC00324=15,686170,169200
BC00325=15,699513,166456
BC00326=15,707199,164860
BC00327=15,702130,176769
BC00328=15,697786,195480
BC00329=15,697786,195480
BC00330=15,703831,213681
BC00331=15,696835,229408
BC00332=302372,698952,211490
BC00333=302372,717858,201268
BC00334=302372,750216,183774
BC00335=305532,747625,53
BC00336=305569,761849,53
BC00337=305584,765283,53
BC00338=305584,756031,53
BC00339=305584,756031,53
BC00340=305584,765283,53
BC00341=305584,765283,53
BC00342=305584,765283,53
BC00343=305584,765283,53
BC00344=305584,765283,53
BC00345=305584,765283,53
BC00346=305584,765283,53
BC00347=242092,730480,4
BC00348=254268,725168,543
BC00349=373423,757548,53
BC00350=374646,771594,53
BC00351=375136,780484,53
BC00352=375136,766039,53
BC00353=375136,766039,53
BC00354=375136,780484,53
BC00355=375136,780484,53
BC00356=326830,797507,51
BC00357=324367,796451,53
BC00358=318212,793809,53
BC00359=331956,796432,138844
BC00360=331956,796432,138844
BC00361=331956,796432,138844
BC00362=331956,796432,138844
BC00363=331956,796432,138844
BC00364=345139,769043,66616
BC00365=345139,804305,66616
BC00366=345139,804305,66616
BC00367=345139,804305,66616
BC00368=345139,804305,66616
BC00369=345139,804305,66616
BC00370=345139,804305,66616
BC00371=345139,804305,66616
BC00372=345139,804305,66616
BC00373=349847,779193,40824
BC00374=390673,737123,107565
BC00375=230273,714746,68332
BC00376=15,702747,12011
BC00377=15,701955,18543
BC00378=15,706339,2244
BC00379=15,708068,108
BC00380=15,708093,53
BC00381=15,708093,53
BC00382=15,708068,108
BC00383=15,708068,108
BC00384=13937,696226,53
BC00385=526,700184,53
BC00386=47,698020,1277
BC00387=766,691948,17562
BC00388=15,702747,12011
BC00389=297950,700262,124402
BC00390=297950,699644,21134
BC00391=369493,695491,225137
BC00392=365725,700831,210595
BC00393=364218,702968,204778
BC00394=364218,702968,204778
BC00395=364218,702968,204778
BC00396=366008,702976,196139
BC00397=367515,700839,201956
BC00398=371283,695499,216499
BC00399=284979,736274,157916
BC00400=281211,741614,143374
BC00401=279704,743751,137557
BC00402=279704,743751,137557
BC00403=279704,743751,137557
BC00404=281466,743758,129052
BC00405=282973,741622,134869
BC00406=286741,736281,149411
BC00407=286720,736279,203179
BC00408=296348,799025,115750
BC00409=298529,835561,48149
BC00410=299550,837400,19199
BC00411=299550,828814,63772
BC00412=299550,828814,63772
BC00413=299550,837400,19199
BC00414=302497,828021,63552
BC00415=297997,829570,63542
BC00416=297997,829570,63542
BC00417=297997,829570,63542
BC00418=297997,829570,63542
BC00419=297997,829570,63542
BC00420=297979,829494,63811
BC00421=296254,822118,90028
BC00422=285994,828831,497
BC00423=289766,832894,53
BC00424=289766,832895,51
BC00425=291275,834519,53
BC00426=291275,834519,53
BC00427=293188,832323,52
BC00428=301226,828160,53
BC00429=301226,828160,53
BC00430=301226,828160,53
BC00431=301226,828160,53
BC00432=301517,827668,53
BC00433=299924,819919,440
BC00434=301049,820896,39095
BC00435=304889,824233,171046
BC00436=304889,700105,171046
BC00437=124585,700105,36
BC00438=124585,700105,36
BC00439=124585,765483,36
BC00440=124585,765483,36
BC00441=124585,765483,36
BC00442=124585,765483,36
BC00443=124585,765483,36
BC00444=124585,765483,36
BC00445=124585,765483,36
BC00446=124585,765483,36
BC00447=124585,765483,36
BC00448=124585,765483,36
BC00449=124585,765483,36
BC00450=124585,765483,36
BC00451=124585,765483,36
BC00452=124585,765483,36
BC00453=124585,765483,36
BC00454=124585,765483,36
BC00455=124585,765483,36
BC00456=124585,765483,36
BC00457=124585,765483,36
BC00458=124585,765483,35
BC00459=124585,765483,35
BC00460=124585,765483,35
BC00461=124585,765483,35
BC00462=124585,765483,35
BC00463=124585,765483,35
BC00464=124585,765483,35
BC00465=124585,765483,35
BC00466=124585,765483,35
BC00467=124585,765483,35
BC00468=124585,765483,35
BC00469=124585,663608,35
BC00470=83775,699365,9536
BC00471=83778,689858,175427
BC00472=83769,691199,148957
BC00473=83766,691735,138369
BC00474=83766,691735,138369
BC00475=83766,691735,138369
BC00476=83766,691735,138369
BC00477=83757,694806,148969
BC00478=83766,693464,175440
BC00479=83763,737347,138110
BC00480=83763,737347,138110
BC00481=197029,737142,72736
BC00482=197039,737143,45852
BC00483=197033,737820,19073
BC00484=197030,738091,8361
BC00485=197030,738091,8361
BC00486=197030,738091,8361
BC00487=197030,738091,8361
BC00488=197021,741431,19085
BC00489=197027,740754,45864
BC00490=196907,776675,45988
BC00491=196900,777352,19209
BC00492=196894,778679,8502
BC00493=196898,777623,8498
BC00494=196898,777623,8498
BC00495=196894,778679,8502
BC00496=196889,780936,19222
BC00497=196895,780259,46001
BC00498=196885,780258,72885
BC00499=171385,775077,62173
BC00500=212214,724112,35449
BC00501=211106,741301,33281
BC00502=211106,741301,33281
BC00503=211368,723652,53
BC00504=211368,723652,53
BC00505=211106,741301,33281
BC00506=208356,721958,8668
BC00507=223868,722216,29649
BC00508=206229,720775,53
BC00509=203870,719461,53
BC00510=202410,718648,52
BC00511=202926,718936,53
BC00512=202926,718936,53
BC00513=202410,718648,52
BC00514=200593,717623,53
BC00515=202951,718937,53
BC00516=191785,744837,53
BC00517=189426,743524,53
BC00518=188187,742833,51
BC00519=188482,742998,53
BC00520=188482,742998,53
BC00521=188187,742833,51
BC00522=186209,741719,53
BC00523=188567,743033,53
BC00524=212591,717178,21939
BC00525=210233,715864,53
BC00526=209289,715339,53
BC00527=209289,715339,53
BC00528=209289,715339,53
BC00529=209289,715339,53
BC00530=206956,714026,53
BC00531=209314,715340,21939
BC00532=192907,721782,82797
BC00533=192907,721782,82797
BC00534=192907,721782,82797
BC00535=192907,721782,82797
BC00536=184359,725138,114504
BC00537=179787,742375,125459
BC00538=167642,738874,171871
BC00539=167642,765336,159298
BC00540=157612,789455,186175
BC00541=157612,789455,186175
BC00542=157612,789455,186175
BC00543=157612,789455,186175
BC00544=157612,789455,186175
BC00545=157612,789455,186175
BC00546=157612,789455,186175
BC00547=157612,789455,186175
BC00548=157612,789455,186175
BC00549=157612,789455,186175
BC00550=157612,789455,186175
BC00551=164113,763380,121188
BC00552=164113,711732,121188
BC00553=279725,698376,1053175
EC00000=798156,0
EC00001=798156,0
EC00002=798156,0
EC00003=798156,0
EC00004=798156,0
EC00005=798156,0
EC00006=798156,0
EC00007=798156,0
EC00008=798156,0
EC00009=798156,0
EC00010=798156,0
EC00011=798156,0
EC00012=798156,0
EC00013=798156,0
EC00014=798156,0
EC00015=798156,0
EC00016=798156,0
EC00017=798156,0
EC00018=798156,0
EC00019=798156,0
EC00020=798156,0
EC00021=798156,0
EC00022=798156,0
EC00023=798156,0
EC00024=798156,0
EC00025=798156,0
EC00026=798156,0
EC00027=798156,0
EC00028=798156,0
EC00029=798156,0
EC00030=798156,0
EC00031=798156,0
EC00032=798156,0
EC00033=798156,0
EC00034=798156,0
EC00035=798156,0
EC00036=798156,0
EC00037=798156,0
EC00038=798156,0
EC00039=798156,0
EC00040=798156,0
EC00041=798156,0
EC00042=798156,0
EC00043=798156,0
EC00044=798156,0
EC00045=798156,0
EC00046=798156,0
EC00047=798156,0
EC00048=798156,0
EC00049=798156,0
EC00050=798156,0
EC00051=798156,0
EC00052=798156,0
EC00053=798156,0
EC00054=798156,0
EC00055=798156,0
EC00056=798156,0
EC00057=798156,0
EC00058=798156,0
EC00059=798156,0
EC00060=798156,0
EC00061=798156,0
EC00062=798156,0
EC00063=798156,0
EC00064=798156,0
EC00065=798156,0
EC00066=798156,0
EC00067=798156,0
EC00068=798156,0
EC00069=798156,0
EC00070=798156,0
EC00071=798156,0
EC00072=798156,0
EC00073=798156,0
EC00074=798156,0
EC00075=798156,0
EC00076=798156,0
EC00077=798156,0
EC00078=798156,0
EC00079=798154,0
EC00080=798156,0
EC00081=798156,0
EC00082=798156,0
EC00083=798156,0
EC00084=798156,0
EC00085=798156,0
EC00086=798156,0
EC00087=798156,0
EC00088=798156,0
EC00089=798156,0
EC00090=798156,0
EC00091=798156,0
EC00092=798156,0
EC00093=798156,0
EC00094=798156,0
EC00095=798156,0
EC00096=798156,0
EC00097=798154,0
EC00098=798154,0
EC00099=798154,0
EC00100=798154,0
EC00101=798154,0
EC00102=798154,0
EC00103=798154,0
EC00104=798154,0
EC00105=798154,0
EC00106=798154,0
EC00107=798154,0
EC00108=798154,0
EC00109=798154,0
EC00110=798154,0
EC00111=798154,0
EC00112=798154,0
EC00113=798154,0
EC00114=798154,0
EC00115=798154,0
EC00116=798154,0
EC00117=798154,0
EC00118=798154,0
EC00119=798154,0
EC00120=798154,0
EC00121=798154,0
EC00122=798154,0
EC00123=798154,0
EC00124=798154,0
EC00125=798154,0
EC00126=798154,0
EC00127=798154,0
EC00128=798154,0
EC00129=798154,0
EC00130=798154,0
EC00131=798154,0
EC00132=798154,0
EC00133=798154,0
EC00134=798154,0
EC00135=798154,0
EC00136=798154,0
EC00137=798154,0
EC00138=798154,0
EC00139=798154,0
EC00140=798154,0
EC00141=798154,0
EC00142=798154,0
EC00143=798154,0
EC00144=798154,0
EC00145=798154,0
EC00146=798154,0
EC00147=798154,0
EC00148=798154,0
EC00149=798154,0
EC00150=798154,0
EC00151=798154,0
EC00152=798154,0
EC00153=798154,0
EC00154=820978,0
EC00155=883374,0
EC00156=975524,0
EC00157=975524,0
EC00158=975524,0
EC00159=975524,0
EC00160=975524,0
EC00161=975524,0
EC00162=975524,0
EC00163=975524,0
EC00164=975524,0
EC00165=975524,0
EC00166=975524,0
EC00167=975524,0
EC00168=975524,0
EC00169=975524,0
EC00170=975524,0
EC00171=975524,0
EC00172=975524,0
EC00173=975524,0
EC00174=975524,0
EC00175=975524,0
EC00176=975524,0
EC00177=975524,0
EC00178=975524,0
EC00179=975524,0
EC00180=975524,0
EC00181=975524,0
EC00182=975524,0
EC00183=975524,0
EC00184=975524,0
EC00185=975524,0
EC00186=975524,0
EC00187=975524,0
EC00188=975524,0
EC00189=975524,0
EC00190=975524,0
EC00191=975524,0
EC00192=975524,0
EC00193=975524,0
EC00194=975524,0
EC00195=975524,0
EC00196=975524,0
EC00197=975524,0
EC00198=975524,0
EC00199=975524,0
EC00200=975524,0
EC00201=975524,0
EC00202=975524,0
EC00203=975524,0
EC00204=975524,0
EC00205=975524,0
EC00206=975524,0
EC00207=975524,0
EC00208=975524,0
EC00209=975524,0
EC00210=975524,0
EC00211=975524,0
EC00212=975524,0
EC00213=975524,0
EC00214=975524,0
EC00215=975524,0
EC00216=975524,0
EC00217=975524,0
EC00218=975524,0
EC00219=975524,0
EC00220=975524,0
EC00221=975524,0
EC00222=975524,0
EC00223=975524,0
EC00224=975524,0
EC00225=975524,0
EC00226=975521,1
EC00227=975523,0
EC00228=975524,0
EC00229=975524,0
EC00230=975524,0
EC00231=975524,0
EC00232=975524,0
EC00233=975524,0
EC00234=975524,0
EC00235=975524,0
EC00236=975524,0
EC00237=975524,0
EC00238=975524,0
EC00239=975521,1
EC00240=975522,0
EC00241=975524,0
EC00242=975524,0
EC00243=975524,0
EC00244=975524,0
EC00245=975524,0
EC00246=975524,0
EC00247=975521,0
EC00248=975524,0
EC00249=975524,0
EC00250=975524,0
EC00251=975524,0
EC00252=975524,0
EC00253=975524,0
EC00254=975524,0
EC00255=975524,0
EC00256=975524,0
EC00257=975524,0
EC00258=975524,0
EC00259=975524,0
EC00260=975524,0
EC00261=975524,0
EC00262=975524,0
EC00263=975524,0
EC00264=975524,0
EC00265=975524,0
EC00266=975524,0
EC00267=975524,0
EC00268=975524,0
EC00269=975524,0
EC00270=975524,0
EC00271=975524,0
EC00272=975524,0
EC00273=975524,0
EC00274=975524,0
EC00275=975524,0
EC00276=975524,0
EC00277=975524,0
EC00278=975524,0
EC00279=975524,0
EC00280=975524,0
EC00281=975524,0
EC00282=975524,0
EC00283=975524,0
EC00284=975524,0
EC00285=975524,0
EC00286=975524,0
EC00287=975524,0
EC00288=975524,0
EC00289=975524,0
EC00290=975524,0
EC00291=975524,0
EC00292=975524,0
EC00293=975524,0
EC00294=975524,0
EC00295=975524,0
EC00296=975524,0
EC00297=975524,0
EC00298=975524,0
EC00299=975524,0
EC00300=975524,0
EC00301=975524,0
EC00302=975524,0
EC00303=975524,0
EC00304=975524,0
EC00305=975524,0
EC00306=975524,0
EC00307=975524,0
EC00308=975524,0
EC00309=975524,0
EC00310=975524,0
EC00311=975524,0
EC00312=975524,0
EC00313=959628,0
EC00314=832192,0
EC00315=798156,0
EC00316=798156,0
EC00317=798156,0
EC00318=798156,0
EC00319=798156,0
EC00320=798156,0
EC00321=798156,0
EC00322=798156,0
EC00323=798156,0
EC00324=798156,0
EC00325=798156,0
EC00326=798156,0
EC00327=798156,0
EC00328=798156,0
EC00329=798156,0
EC00330=798156,0
EC00331=798156,0
EC00332=798156,0
EC00333=798156,0
EC00334=798156,0
EC00335=798156,0
EC00336=798156,0
EC00337=798156,0
EC00338=798156,0
EC00339=798156,0
EC00340=798156,0
EC00341=798156,0
EC00342=798156,0
EC00343=798156,0
EC00344=798156,0
EC00345=798156,0
EC00346=798156,0
EC00347=798156,0
EC00348=798156,0
EC00349=798156,0
EC00350=798156,0
EC00351=798156,0
EC00352=798156,0
EC00353=798156,0
EC00354=798156,0
EC00355=798156,0
EC00356=798154,1
EC00357=798156,0
EC00358=798156,0
EC00359=798156,0
EC00360=798156,0
EC00361=798156,0
EC00362=798156,0
EC00363=798156,0
EC00364=798156,0
EC00365=798156,0
EC00366=798156,0
EC00367=798156,0
EC00368=798156,0
EC00369=798156,0
EC00370=798156,0
EC00371=798156,0
EC00372=798156,0
EC00373=798156,0
EC00374=798156,0
EC00375=798156,0
EC00376=798156,0
EC00377=798156,0
EC00378=798156,0
EC00379=798156,0
EC00380=798156,0
EC00381=798156,0
EC00382=798156,0
EC00383=798156,0
EC00384=798156,0
EC00385=798156,0
EC00386=798156,0
EC00387=798156,0
EC00388=798156,0
EC00389=798156,0
EC00390=798156,0
EC00391=798156,0
EC00392=798156,0
EC00393=798156,0
EC00394=798156,0
EC00395=798156,0
EC00396=798156,0
EC00397=798156,0
EC00398=798156,0
EC00399=798156,0
EC00400=798156,0
EC00401=798156,0
EC00402=798156,0
EC00403=798156,0
EC00404=798156,0
EC00405=798156,0
EC00406=798156,0
EC00407=798156,0
EC00408=798156,0
EC00409=798156,0
EC00410=798156,0
EC00411=798156,0
EC00412=798156,0
EC00413=798156,0
EC00414=798156,0
EC00415=798155,1
EC00416=798155,1
EC00417=798155,1
EC00418=798155,1
EC00419=798155,1
EC00420=798155,1
EC00421=798156,0
EC00422=798156,0
EC00423=798156,0
EC00424=798155,0
EC00425=798156,0
EC00426=798156,0
EC00427=798156,0
EC00428=798156,0
EC00429=798156,0
EC00430=798156,0
EC00431=798156,0
EC00432=798156,0
EC00433=798156,0
EC00434=798156,0
EC00435=798156,0
EC00436=798156,0
EC00437=798156,0
EC00438=798156,0
EC00439=798156,0
EC00440=798156,0
EC00441=798156,0
EC00442=798156,0
EC00443=798156,0
EC00444=798156,0
EC00445=798156,0
EC00446=798156,0
EC00447=798156,0
EC00448=798156,0
EC00449=798156,0
EC00450=798156,0
EC00451=798156,0
EC00452=798156,0
EC00453=798156,0
EC00454=798156,0
EC00455=798156,0
EC00456=798156,0
EC00457=798156,0
EC00458=798155,1
EC00459=798155,1
EC00460=798155,1
EC00461=798155,1
EC00462=798155,1
EC00463=798155,1
EC00464=798155,1
EC00465=798155,1
EC00466=798155,1
EC00467=798155,1
EC00468=798155,1
EC00469=798155,1
EC00470=798156,0
EC00471=798156,0
EC00472=798156,0
EC00473=798156,0
EC00474=798156,0
EC00475=798156,0
EC00476=798156,0
EC00477=798156,0
EC00478=798156,0
EC00479=798156,0
EC00480=798156,0
EC00481=798156,0
EC00482=798156,0
EC00483=798156,0
EC00484=798156,0
EC00485=798156,0
EC00486=798156,0
EC00487=798156,0
EC00488=798156,0
EC00489=798156,0
EC00490=798156,0
EC00491=798156,0
EC00492=798156,0
EC00493=798156,0
EC00494=798156,0
EC00495=798156,0
EC00496=798156,0
EC00497=798156,0
EC00498=798156,0
EC00499=798156,0
EC00500=798156,0
EC00501=798156,0
EC00502=798156,0
EC00503=798156,0
EC00504=798156,0
EC00505=798156,0
EC00506=798156,0
EC00507=798156,0
EC00508=798156,0
EC00509=798156,0
EC00510=798155,0
EC00511=798156,0
EC00512=798156,0
EC00513=798155,0
EC00514=798156,0
EC00515=798156,0
EC00516=798156,0
EC00517=798156,0
EC00518=798154,1
EC00519=798156,0
EC00520=798156,0
EC00521=798154,1
EC00522=798156,0
EC00523=798156,0
EC00524=798156,0
EC00525=798156,0
EC00526=798156,0
EC00527=798156,0
EC00528=798156,0
EC00529=798156,0
EC00530=798156,0
EC00531=798156,0
EC00532=798156,0
EC00533=798156,0
EC00534=798156,0
EC00535=798156,0
EC00536=798156,0
EC00537=798156,0
EC00538=798156,0
EC00539=798156,0
EC00540=798156,0
EC00541=798156,0
EC00542=798156,0
EC00543=798156,0
EC00544=798156,0
EC00545=798156,0
EC00546=798156,0
EC00547=798156,0
EC00548=798156,0
EC00549=798156,0
EC00550=798156,0
EC00551=798156,0
EC00552=798156,0
EC00553=798156,0
///POSTYPE BASE
///RECTAN
///RCONF 0,0,0,0,0,0,0,0,0,0,0,0,0,0,0,0,0,0,0,0,0,0,0,0
P00006=0.222,-3.123,-1.508,0.0000,0.0000,0.0000
P00021=-0.225,-6.128,-0.405,0.0000,0.0000,0.0000
P00022=0.222,-3.123,-1.508,0.0000,0.0000,0.0000
P00024=0.145,-0.552,1.326,0.0000,0.0000,0.0000
P00025=-2.003,0.006,0.728,0.0000,0.0000,0.0000
P00026=0.562,-0.002,-0.337,0.0000,0.0000,0.0000
P00027=-0.746,0.015,-9.096,0.0000,0.0000,0.0000
P00032=1.957,0.503,-7.217,0.0000,0.0000,0.0000
P00041=0.192,3.924,0.305,0.0000,0.0000,0.0000
P00042=-0.217,1.941,0.413,0.0000,0.0000,0.0000
P00043=-0.044,-1.937,1.197,0.0000,0.0000,0.0000
P00044=0.687,-2.322,1.156,0.0000,0.0000,0.0000
P00045=-0.068,-0.810,1.603,0.0000,0.0000,0.0000
P00046=0.799,0.043,1.292,0.0000,0.0000,0.0000
P00051=0.367,3.892,0.009,0.0000,0.0000,0.0000
P00052=0.088,2.832,-0.342,0.0000,0.0000,0.0000
P00053=0.134,6.594,0.107,0.0000,0.0000,0.0000
P00054=-0.103,6.509,-0.702,0.0000,0.0000,0.0000
P00055=-0.342,8.912,1.324,0.0000,0.0000,0.0000
P00056=0.568,-0.032,0.830,0.0000,0.0000,0.0000
P00066=5.557,-0.028,3.115,0.0000,0.0000,0.0000
///RCONF 0,1,0,0,0,0,0,0,0,0,0,0,0,0,0,0,0,0,0,0,0,0,0,0
P00067=-0.081,0.026,-1.119,0.0000,0.0000,0.0000
///RCONF 0,0,0,0,0,0,0,0,0,0,0,0,0,0,0,0,0,0,0,0,0,0,0,0
P00068=2.896,1.192,4.622,0.0000,0.0000,0.0000
//INST
///DATE 2025/01/29 14:24
///ATTR SC,RW
///GROUP1 RB1,BS1
///GROUP2 ST1
NOP
'OK_r2_O57-69(1)(90,0)
'Down
'Path S1900
SFTOF3D
'Path S1901
SFTOF3D
MOVJ C00000 BC00000 VJ=40.00  +MOVJ EC00000 VJ=15.00
MOVJ C00001 BC00001 VJ=100.00  +MOVJ EC00001 VJ=100.00
MOVL C00002 BC00002 V=400.0  +MOVJ EC00002 VJ=100.00
SMOVL C00003 BC00003 V=100.0  +MOVJ EC00003
SREFP 3 C00004 BC00004  +REFP EC00004
CALL JOB:SEARCH-R1-S13D
SET P026 P006
SFTON3D P026
SMOVL C00005 BC00005 V=100.0  +MOVJ EC00005
SREFP 3 C00006 BC00006  +REFP EC00006
CALL JOB:SEARCH-R1-S13D
SET P026 P006
SFTON3D P026
SMOVL C00007 BC00007 V=100.0  +MOVJ EC00007
MOVL C00008 BC00008 V=400.0  +MOVJ EC00008 VJ=100.00
MOVL C00009 BC00009 V=1000.0  +MOVJ EC00009 VJ=100.00
'Path S1902
SFTOF3D
MOVJ C00010 BC00010 VJ=100.00  +MOVJ EC00010 VJ=100.00
MOVL C00011 BC00011 V=400.0  +MOVJ EC00011 VJ=100.00
SMOVL C00012 BC00012 V=100.0  +MOVJ EC00012
SREFP 3 C00013 BC00013  +REFP EC00013
CALL JOB:SEARCH-R1-S13D
SET P027 P006
SFTON3D P027
SMOVL C00014 BC00014 V=100.0  +MOVJ EC00014
SREFP 3 C00015 BC00015  +REFP EC00015
CALL JOB:SEARCH-R1-S13D
SET P027 P006
SFTON3D P027
SMOVL C00016 BC00016 V=100.0  +MOVJ EC00016
SFTOF3D
MOVL C00017 BC00017 V=400.0  +MOVJ EC00017 VJ=100.00
MOVL C00018 BC00018 V=1000.0  +MOVJ EC00018 VJ=100.00
MOVJ C00019 BC00019 VJ=100.00  +MOVJ EC00019 VJ=100.00
'Path S1903
SFTOF3D
MOVJ C00020 BC00020 VJ=100.00  +MOVJ EC00020 VJ=100.00
COMM PAUSE
COMM MOVL C00021 BC00021 V=400.0  +MOVJ EC00021 VJ=100.00
COMM SMOVL C00022 BC00022 V=100.0  +MOVJ EC00022
COMM SREFP 3 C00023 BC00023  +REFP EC00023
COMM CALL JOB:SEARCH-R1-S13D
COMM SET P022 P006
COMM SFTON3D P022
COMM SMOVL C00024 BC00024 V=100.0  +MOVJ EC00024
COMM SREFP 3 C00025 BC00025  +REFP EC00025
COMM CALL JOB:SEARCH-R1-S13D
COMM SET P022 P006
COMM SFTON3D P022
COMM SMOVL C00026 BC00026 V=100.0  +MOVJ EC00026
COMM SFTOF3D
COMM MOVL C00027 BC00027 V=400.0  +MOVJ EC00027 VJ=100.00
MOVL C00028 BC00028 V=1000.0  +MOVJ EC00028 VJ=100.00
SMOVL C00029 BC00029 V=1000.0  +MOVJ EC00029
SMOVL C00030 BC00030 V=1000.0  +MOVJ EC00030
SMOVL C00031 BC00031 V=166.7  +MOVJ EC00031
SREFP 3 C00032 BC00032  +REFP EC00032
CALL JOB:SEARCH-R1-S13D
SET P066 P006
SFTON3D P066
SMOVL C00033 BC00033 V=250.0  +MOVJ EC00033
SMOVL C00034 BC00034 V=250.0  +MOVJ EC00034
SMOVL C00035 BC00035 V=250.0  +MOVJ EC00035
SREFP 3 C00036 BC00036  +REFP EC00036
CALL JOB:SEARCH-R1-S13D
SET P066 P006
SFTON3D P066
SMOVL C00037 BC00037 V=250.0  +MOVJ EC00037
SMOVL C00038 BC00038 V=1000.0  +MOVJ EC00038
SFTOF3D
SMOVL C00039 BC00039 V=1000.0  +MOVJ EC00039
SMOVL C00040 BC00040 V=166.7  +MOVJ EC00040
SREFP 3 C00041 BC00041  +REFP EC00041
CALL JOB:SEARCH-R1-S13D
SET P068 P006
SFTON3D P068
SMOVL C00042 BC00042 V=250.0  +MOVJ EC00042
SREFP 3 C00043 BC00043  +REFP EC00043
CALL JOB:SEARCH-R1-S13D
SET P068 P006
SFTON3D P068
SMOVL C00044 BC00044 V=250.0  +MOVJ EC00044
SMOVL C00045 BC00045 V=166.7  +MOVJ EC00045
SREFP 3 C00046 BC00046  +REFP EC00046
CALL JOB:SEARCH-R1-S13D
SET P068 P006
SFTON3D P068
SMOVL C00047 BC00047 V=250.0  +MOVJ EC00047
SFTOF3D
SMOVL C00048 BC00048 V=1000.0  +MOVJ EC00048
MOVJ C00049 BC00049 VJ=100.00  +MOVJ EC00049 VJ=100.00
MOVJ C00050 BC00050 VJ=100.00  +MOVJ EC00050 VJ=100.00
COMM PAUSE
COMM MOVJ C00051 BC00051 VJ=100.00  +MOVJ EC00051 VJ=100.00
COMM SMOVL C00052 BC00052 V=1000.0  +MOVJ EC00052
COMM SMOVL C00053 BC00053 V=166.7  +MOVJ EC00053
COMM SREFP 3 C00054 BC00054  +REFP EC00054
COMM CALL JOB:SEARCH-R1-S13D
COMM SET P067 P006
COMM SFTON3D P067
COMM SMOVL C00055 BC00055 V=250.0  +MOVJ EC00055
COMM SMOVL C00056 BC00056 V=250.0  +MOVJ EC00056
COMM SMOVL C00057 BC00057 V=133.3  +MOVJ EC00057
COMM SREFP 3 C00058 BC00058  +REFP EC00058
COMM CALL JOB:SEARCH-R1-S13D
COMM SET P067 P006
COMM SFTON3D P067
COMM SMOVL C00059 BC00059 V=250.0  +MOVJ EC00059
COMM SFTOF3D
COMM SMOVL C00060 BC00060 V=1000.0  +MOVJ EC00060
SMOVL C00061 BC00061 V=1000.0  +MOVJ EC00061
MOVJ C00062 BC00062 VJ=100.00  +MOVJ EC00062 VJ=50.00
MOVJ C00063 BC00063 VJ=100.00  +MOVJ EC00063 VJ=100.00
MOVL C00064 BC00064 V=400.0  +MOVJ EC00064 VJ=100.00
SMOVL C00065 BC00065 V=100.0  +MOVJ EC00065
SREFP 3 C00066 BC00066  +REFP EC00066
CALL JOB:SEARCH-R1-S13D
SET P021 P006
SFTON3D P021
SMOVL C00067 BC00067 V=100.0  +MOVJ EC00067
SMOVL C00068 BC00068 V=100.0  +MOVJ EC00068
SREFP 3 C00069 BC00069  +REFP EC00069
CALL JOB:SEARCH-R1-S13D
SET P021 P006
SFTON3D P021
SMOVL C00070 BC00070 V=100.0  +MOVJ EC00070
SMOVL C00071 BC00071 V=100.0  +MOVJ EC00071
SREFP 3 C00072 BC00072  +REFP EC00072
CALL JOB:SEARCH-R1-S13D
SET P021 P006
SFTON3D P021
SMOVL C00073 BC00073 V=100.0  +MOVJ EC00073
MOVL C00074 BC00074 V=400.0  +MOVJ EC00074 VJ=100.00
MOVL C00075 BC00075 V=1000.0  +MOVJ EC00075 VJ=100.00
MOVJ C00076 BC00076 VJ=100.00  +MOVJ EC00076 VJ=100.00
MOVJ C00077 BC00077 VJ=100.00  +MOVJ EC00077 VJ=100.00
MOVJ C00078 BC00078 VJ=100.00  +MOVJ EC00078 VJ=100.00
MOVJ C00079 BC00079 VJ=100.00  +MOVJ EC00079 VJ=100.00
'Path S1912
SFTOF3D
MOVJ C00080 BC00080 VJ=100.00  +MOVJ EC00080 VJ=100.00
MOVL C00081 BC00081 V=400.0  +MOVJ EC00081 VJ=100.00
SMOVL C00082 BC00082 V=100.0  +MOVJ EC00082
SREFP 3 C00083 BC00083  +REFP EC00083
CALL JOB:SEARCH-R1-S13D
SET P032 P006
SFTON3D P032
SMOVL C00084 BC00084 V=100.0  +MOVJ EC00084
SMOVL C00085 BC00085 V=100.0  +MOVJ EC00085
SREFP 3 C00086 BC00086  +REFP EC00086
CALL JOB:SEARCH-R1-S13D
SET P032 P006
SFTON3D P032
SMOVL C00087 BC00087 V=100.0  +MOVJ EC00087
SFTOF3D
MOVL C00088 BC00088 V=400.0  +MOVJ EC00088 VJ=100.00
MOVL C00089 BC00089 V=1000.0  +MOVJ EC00089 VJ=100.00
MOVJ C00090 BC00090 VJ=100.00  +MOVJ EC00090 VJ=100.00
MOVJ C00091 BC00091 VJ=100.00  +MOVJ EC00091 VJ=100.00
'Up
MOVJ C00092 BC00092 VJ=100.00  +MOVJ EC00092 VJ=50.00
MOVJ C00093 BC00093 VJ=100.00  +MOVJ EC00093 VJ=100.00
MOVJ C00094 BC00094 VJ=100.00  +MOVJ EC00094 VJ=100.00
MOVJ C00095 BC00095 VJ=100.00  +MOVJ EC00095 VJ=100.00
SMOVL C00096 BC00096 V=666.7  +MOVJ EC00096
SMOVL C00097 BC00097 V=166.7  +MOVJ EC00097
SREFP 3 C00098 BC00098  +REFP EC00098
CALL JOB:SEARCH-R1-S13D
SET P051 P006
SFTON3D P051
SMOVL C00099 BC00099 V=166.7  +MOVJ EC00099
SMOVL C00100 BC00100 V=166.7  +MOVJ EC00100
SMOVL C00101 BC00101 V=166.7  +MOVJ EC00101
SREFP 3 C00102 BC00102  +REFP EC00102
CALL JOB:SEARCH-R1-S13D
SET P051 P006
SFTON3D P051
SMOVL C00103 BC00103 V=166.7  +MOVJ EC00103
SMOVL C00104 BC00104 V=666.7  +MOVJ EC00104
SMOVL C00105 BC00105 V=166.7  +MOVJ EC00105
SREFP 3 C00106 BC00106  +REFP EC00106
CALL JOB:SEARCH-R1-S13D
SET P051 P006
SFTON3D P051
SMOVL C00107 BC00107 V=166.7  +MOVJ EC00107
SMOVL C00108 BC00108 V=166.7  +MOVJ EC00108
SMOVL C00109 BC00109 V=166.7  +MOVJ EC00109
SREFP 3 C00110 BC00110  +REFP EC00110
CALL JOB:SEARCH-R1-S13D
SET P051 P006
SFTON3D P051
SMOVL C00111 BC00111 V=166.7  +MOVJ EC00111
SMOVL C00112 BC00112 V=666.7  +MOVJ EC00112
SMOVL C00113 BC00113 V=166.7  +MOVJ EC00113
SREFP 3 C00114 BC00114  +REFP EC00114
CALL JOB:SEARCH-R1-S13D
SET P052 P006
SFTON3D P052
SMOVL C00115 BC00115 V=166.7  +MOVJ EC00115
SMOVL C00116 BC00116 V=166.7  +MOVJ EC00116
SMOVL C00117 BC00117 V=166.7  +MOVJ EC00117
SREFP 3 C00118 BC00118  +REFP EC00118
CALL JOB:SEARCH-R1-S13D
SET P052 P006
SFTON3D P052
SMOVL C00119 BC00119 V=166.7  +MOVJ EC00119
SMOVL C00120 BC00120 V=666.7  +MOVJ EC00120
SMOVL C00121 BC00121 V=166.7  +MOVJ EC00121
SREFP 3 C00122 BC00122  +REFP EC00122
CALL JOB:SEARCH-R1-S13D
SET P053 P006
SFTON3D P053
SMOVL C00123 BC00123 V=166.7  +MOVJ EC00123
SMOVL C00124 BC00124 V=166.7  +MOVJ EC00124
SMOVL C00125 BC00125 V=166.7  +MOVJ EC00125
SREFP 3 C00126 BC00126  +REFP EC00126
CALL JOB:SEARCH-R1-S13D
SET P053 P006
SFTON3D P053
SMOVL C00127 BC00127 V=166.7  +MOVJ EC00127
SMOVL C00128 BC00128 V=666.7  +MOVJ EC00128
SMOVL C00129 BC00129 V=166.7  +MOVJ EC00129
SREFP 3 C00130 BC00130  +REFP EC00130
CALL JOB:SEARCH-R1-S13D
SET P054 P006
SFTON3D P054
SMOVL C00131 BC00131 V=166.7  +MOVJ EC00131
SMOVL C00132 BC00132 V=166.7  +MOVJ EC00132
SMOVL C00133 BC00133 V=166.7  +MOVJ EC00133
SREFP 3 C00134 BC00134  +REFP EC00134
CALL JOB:SEARCH-R1-S13D
SET P054 P006
SFTON3D P054
SMOVL C00135 BC00135 V=166.7  +MOVJ EC00135
SMOVL C00136 BC00136 V=666.7  +MOVJ EC00136
SMOVL C00137 BC00137 V=166.7  +MOVJ EC00137
SREFP 3 C00138 BC00138  +REFP EC00138
CALL JOB:SEARCH-R1-S13D
SET P055 P006
SFTON3D P055
SMOVL C00139 BC00139 V=166.7  +MOVJ EC00139
SMOVL C00140 BC00140 V=166.7  +MOVJ EC00140
SMOVL C00141 BC00141 V=166.7  +MOVJ EC00141
SREFP 3 C00142 BC00142  +REFP EC00142
CALL JOB:SEARCH-R1-S13D
SET P055 P006
SFTON3D P055
SMOVL C00143 BC00143 V=166.7  +MOVJ EC00143
SMOVL C00144 BC00144 V=666.7  +MOVJ EC00144
SMOVL C00145 BC00145 V=166.7  +MOVJ EC00145
SREFP 3 C00146 BC00146  +REFP EC00146
CALL JOB:SEARCH-R1-S13D
SET P056 P006
SFTON3D P056
SMOVL C00147 BC00147 V=166.7  +MOVJ EC00147
SMOVL C00148 BC00148 V=166.7  +MOVJ EC00148
SMOVL C00149 BC00149 V=166.7  +MOVJ EC00149
SREFP 3 C00150 BC00150  +REFP EC00150
CALL JOB:SEARCH-R1-S13D
SET P056 P006
SFTON3D P056
SMOVL C00151 BC00151 V=166.7  +MOVJ EC00151
SFTOF3D
MOVL C00152 BC00152 V=666.7  +MOVJ EC00152 VJ=100.00
MOVL C00153 BC00153 V=666.7  +MOVJ EC00153 VJ=100.00
MOVJ C00154 BC00154 VJ=100.00  +MOVJ EC00154 VJ=100.00
MOVJ C00155 BC00155 VJ=100.00  +MOVJ EC00155 VJ=100.00
MOVJ C00156 BC00156 VJ=100.00  +MOVJ EC00156 VJ=100.00
MOVJ C00157 BC00157 VJ=100.00  +MOVJ EC00157 VJ=100.00
'Path S1137
SFTOF3D
MOVJ C00158 BC00158 VJ=100.00  +MOVJ EC00158 VJ=100.00
MOVL C00159 BC00159 V=400.0  +MOVJ EC00159 VJ=100.00
SMOVL C00160 BC00160 V=100.0  +MOVJ EC00160
SREFP 3 C00161 BC00161  +REFP EC00161
CALL JOB:SEARCH-R1-S13D
SET P046 P006
SFTON3D P046
SMOVL C00162 BC00162 V=100.0  +MOVJ EC00162
SMOVL C00163 BC00163 V=100.0  +MOVJ EC00163
SREFP 3 C00164 BC00164  +REFP EC00164
CALL JOB:SEARCH-R1-S13D
SET P046 P006
SFTON3D P046
SMOVL C00165 BC00165 V=100.0  +MOVJ EC00165
MOVL C00166 BC00166 V=400.0  +MOVJ EC00166 VJ=100.00
MOVL C00167 BC00167 V=1000.0  +MOVJ EC00167 VJ=100.00
'Path S1169
SFTOF3D
MOVJ C00168 BC00168 VJ=100.00  +MOVJ EC00168 VJ=100.00
MOVL C00169 BC00169 V=400.0  +MOVJ EC00169 VJ=100.00
SMOVL C00170 BC00170 V=100.0  +MOVJ EC00170
SREFP 3 C00171 BC00171  +REFP EC00171
CALL JOB:SEARCH-R1-S13D
SET P045 P006
SFTON3D P045
SMOVL C00172 BC00172 V=100.0  +MOVJ EC00172
SREFP 3 C00173 BC00173  +REFP EC00173
CALL JOB:SEARCH-R1-S13D
SET P045 P006
SFTON3D P045
SMOVL C00174 BC00174 V=100.0  +MOVJ EC00174
SREFP 3 C00175 BC00175  +REFP EC00175
CALL JOB:SEARCH-R1-S13D
SET P045 P006
SFTON3D P045
SMOVL C00176 BC00176 V=100.0  +MOVJ EC00176
SFTOF3D
MOVL C00177 BC00177 V=400.0  +MOVJ EC00177 VJ=100.00
MOVL C00178 BC00178 V=1000.0  +MOVJ EC00178 VJ=100.00
MOVL C00179 BC00179 V=1000.0  +MOVJ EC00179 VJ=100.00
MOVJ C00180 BC00180 VJ=100.00  +MOVJ EC00180 VJ=50.00
MOVJ C00181 BC00181 VJ=100.00  +MOVJ EC00181 VJ=50.00
MOVJ C00182 BC00182 VJ=100.00  +MOVJ EC00182 VJ=100.00
MOVL C00183 BC00183 V=400.0  +MOVJ EC00183 VJ=100.00
SMOVL C00184 BC00184 V=100.0  +MOVJ EC00184
SREFP 3 C00185 BC00185  +REFP EC00185
CALL JOB:SEARCH-R1-S13D
SET P043 P006
SFTON3D P043
SMOVL C00186 BC00186 V=100.0  +MOVJ EC00186
SMOVL C00187 BC00187 V=100.0  +MOVJ EC00187
SREFP 3 C00188 BC00188  +REFP EC00188
CALL JOB:SEARCH-R1-S13D
SET P043 P006
SFTON3D P043
SMOVL C00189 BC00189 V=100.0  +MOVJ EC00189
SMOVL C00190 BC00190 V=100.0  +MOVJ EC00190
SREFP 3 C00191 BC00191  +REFP EC00191
CALL JOB:SEARCH-R1-S13D
SET P043 P006
SFTON3D P043
SMOVL C00192 BC00192 V=100.0  +MOVJ EC00192
MOVL C00193 BC00193 V=400.0  +MOVJ EC00193 VJ=100.00
MOVL C00194 BC00194 V=1000.0  +MOVJ EC00194 VJ=100.00
'Path S1166
SFTOF3D
MOVJ C00195 BC00195 VJ=100.00  +MOVJ EC00195 VJ=100.00
MOVL C00196 BC00196 V=400.0  +MOVJ EC00196 VJ=100.00
SMOVL C00197 BC00197 V=100.0  +MOVJ EC00197
SREFP 3 C00198 BC00198  +REFP EC00198
CALL JOB:SEARCH-R1-S13D
SET P042 P006
SFTON3D P042
SMOVL C00199 BC00199 V=100.0  +MOVJ EC00199
SMOVL C00200 BC00200 V=100.0  +MOVJ EC00200
SREFP 3 C00201 BC00201  +REFP EC00201
CALL JOB:SEARCH-R1-S13D
SET P042 P006
SFTON3D P042
SMOVL C00202 BC00202 V=100.0  +MOVJ EC00202
SMOVL C00203 BC00203 V=100.0  +MOVJ EC00203
SREFP 3 C00204 BC00204  +REFP EC00204
CALL JOB:SEARCH-R1-S13D
SET P042 P006
SFTON3D P042
SMOVL C00205 BC00205 V=100.0  +MOVJ EC00205
MOVL C00206 BC00206 V=400.0  +MOVJ EC00206 VJ=100.00
MOVL C00207 BC00207 V=1000.0  +MOVJ EC00207 VJ=100.00
'Path S1165
SFTOF3D
MOVJ C00208 BC00208 VJ=100.00  +MOVJ EC00208 VJ=100.00
MOVL C00209 BC00209 V=400.0  +MOVJ EC00209 VJ=100.00
SMOVL C00210 BC00210 V=100.0  +MOVJ EC00210
SREFP 3 C00211 BC00211  +REFP EC00211
CALL JOB:SEARCH-R1-S13D
SET P041 P006
SFTON3D P041
SMOVL C00212 BC00212 V=100.0  +MOVJ EC00212
SMOVL C00213 BC00213 V=100.0  +MOVJ EC00213
SREFP 3 C00214 BC00214  +REFP EC00214
CALL JOB:SEARCH-R1-S13D
SET P041 P006
SFTON3D P041
SMOVL C00215 BC00215 V=100.0  +MOVJ EC00215
SMOVL C00216 BC00216 V=100.0  +MOVJ EC00216
SREFP 3 C00217 BC00217  +REFP EC00217
CALL JOB:SEARCH-R1-S13D
SET P041 P006
SFTON3D P041
SMOVL C00218 BC00218 V=100.0  +MOVJ EC00218
MOVL C00219 BC00219 V=400.0  +MOVJ EC00219 VJ=100.00
MOVL C00220 BC00220 V=1000.0  +MOVJ EC00220 VJ=100.00
'Path W378
SFTOF3D
SFTON3D P041
MOVJ C00221 BC00221 VJ=100.00  +MOVJ EC00221 VJ=100.00
SMOVL C00222 BC00222 V=400.0  +MOVJ EC00222
SMOVL C00223 BC00223 V=133.3 PL=0  +MOVJ EC00223
SREFP 1 C00224 BC00224  +REFP EC00224
SREFP 2 C00225 BC00225  +REFP EC00225
MACRO1 MJ#(0) ARGF9
ARCON
SWVON WEV#(61)
SMOVL C00226 BC00226 V=6.7  +MOVJ EC00226
SMOVL C00227 BC00227 V=6.7  +MOVJ EC00227
SMOVL C00228 BC00228 V=6.7  +MOVJ EC00228
ARCOF
SWVOF
SMOVL C00229 BC00229 V=400.0  +MOVJ EC00229
SMOVL C00230 BC00230 V=1000.0  +MOVJ EC00230
SFTOF3D
MOVJ C00231 BC00231 VJ=100.00  +MOVJ EC00231 VJ=100.00
'Path W379
SFTOF3D
SFTON3D P042
MOVJ C00232 BC00232 VJ=100.00  +MOVJ EC00232 VJ=100.00
MOVJ C00233 BC00233 VJ=100.00  +MOVJ EC00233 VJ=100.00
SMOVL C00234 BC00234 V=400.0  +MOVJ EC00234
SMOVL C00235 BC00235 V=133.3 PL=0  +MOVJ EC00235
SREFP 1 C00236 BC00236  +REFP EC00236
SREFP 2 C00237 BC00237  +REFP EC00237
MACRO1 MJ#(0) ARGF9
ARCON
SMOVL C00238 BC00238 V=9.2  +MOVJ EC00238
SMOVL C00239 BC00239 V=9.2  +MOVJ EC00239
SMOVL C00240 BC00240 V=9.2  +MOVJ EC00240
ARCOF
SMOVL C00241 BC00241 V=400.0  +MOVJ EC00241
SMOVL C00242 BC00242 V=1000.0  +MOVJ EC00242
SFTOF3D
MOVJ C00243 BC00243 VJ=20.00  +MOVJ EC00243 VJ=100.00
'Path W380
SFTOF3D
SFTON3D P043
MOVJ C00244 BC00244 VJ=100.00  +MOVJ EC00244 VJ=100.00
MOVJ C00245 BC00245 VJ=100.00  +MOVJ EC00245 VJ=100.00
SMOVL C00246 BC00246 V=400.0  +MOVJ EC00246
SMOVL C00247 BC00247 V=133.3 PL=0  +MOVJ EC00247
SREFP 1 C00248 BC00248  +REFP EC00248
SREFP 2 C00249 BC00249  +REFP EC00249
ARCON
SMOVL C00250 BC00250 V=9.2  +MOVJ EC00250
SMOVL C00251 BC00251 V=9.2  +MOVJ EC00251
ARCOF
SMOVL C00252 BC00252 V=400.0  +MOVJ EC00252
SMOVL C00253 BC00253 V=1000.0  +MOVJ EC00253
SMOVL C00254 BC00254 V=1000.0  +MOVJ EC00254
MOVJ C00255 BC00255 VJ=100.00  +MOVJ EC00255 VJ=100.00
SFTOF3D
'NIE SPAWAMY
COMM 'Path W381
COMM SFTOF3D
COMM SFTON3D P044
COMM MOVJ C00256 BC00256 VJ=100.00  +MOVJ EC00256 VJ=100.00
COMM SMOVL C00257 BC00257 V=400.0  +MOVJ EC00257
COMM SMOVL C00258 BC00258 V=100.0 PL=0  +MOVJ EC00258
COMM SREFP 1 C00259 BC00259  +REFP EC00259
COMM SREFP 2 C00260 BC00260  +REFP EC00260
COMM MACRO1 MJ#(0) ARGF0
COMM ARCON
COMM SMOVL C00261 BC00261 V=10.0  +MOVJ EC00261
COMM SMOVL C00262 BC00262 V=10.0  +MOVJ EC00262
COMM SMOVL C00263 BC00263 V=10.0  +MOVJ EC00263
COMM SMOVL C00264 BC00264 V=10.0  +MOVJ EC00264
COMM SMOVL C00265 BC00265 V=10.0  +MOVJ EC00265
COMM SMOVL C00266 BC00266 V=10.0  +MOVJ EC00266
COMM SMOVL C00267 BC00267 V=10.0  +MOVJ EC00267
COMM SMOVL C00268 BC00268 V=10.0  +MOVJ EC00268
COMM SMOVL C00269 BC00269 V=10.0  +MOVJ EC00269
COMM SMOVL C00270 BC00270 V=10.0  +MOVJ EC00270
COMM SMOVL C00271 BC00271 V=10.0  +MOVJ EC00271
COMM SMOVL C00272 BC00272 V=10.0  +MOVJ EC00272
COMM SMOVL C00273 BC00273 V=10.0  +MOVJ EC00273
COMM SMOVL C00274 BC00274 V=10.0  +MOVJ EC00274
COMM SMOVL C00275 BC00275 V=10.0  +MOVJ EC00275
COMM SMOVL C00276 BC00276 V=10.0  +MOVJ EC00276
COMM SMOVL C00277 BC00277 V=10.0  +MOVJ EC00277
COMM SMOVL C00278 BC00278 V=10.0  +MOVJ EC00278
COMM SMOVL C00279 BC00279 V=10.0  +MOVJ EC00279
COMM SMOVL C00280 BC00280 V=10.0  +MOVJ EC00280
COMM SMOVL C00281 BC00281 V=10.0  +MOVJ EC00281
COMM SMOVL C00282 BC00282 V=10.0  +MOVJ EC00282
COMM SMOVL C00283 BC00283 V=10.0  +MOVJ EC00283
COMM SMOVL C00284 BC00284 V=10.0  +MOVJ EC00284
COMM SMOVL C00285 BC00285 V=10.0  +MOVJ EC00285
COMM ARCOF
COMM SMOVL C00286 BC00286 V=400.0  +MOVJ EC00286
COMM SMOVL C00287 BC00287 V=1000.0  +MOVJ EC00287
COMM SFTOF3D
'Path W382
SFTOF3D
MOVJ C00288 BC00288 VJ=100.00  +MOVJ EC00288 VJ=50.00
SFTON3D P045
MOVJ C00289 BC00289 VJ=100.00  +MOVJ EC00289 VJ=100.00
SMOVL C00290 BC00290 V=400.0  +MOVJ EC00290
SMOVL C00291 BC00291 V=133.3 PL=0  +MOVJ EC00291
SREFP 1 C00292 BC00292  +REFP EC00292
SREFP 2 C00293 BC00293  +REFP EC00293
ARCON
SMOVL C00294 BC00294 V=9.2  +MOVJ EC00294
SMOVL C00295 BC00295 V=9.2  +MOVJ EC00295
SMOVL C00296 BC00296 V=9.2  +MOVJ EC00296
ARCOF
SMOVL C00297 BC00297 V=400.0  +MOVJ EC00297
SMOVL C00298 BC00298 V=1000.0  +MOVJ EC00298
SMOVL C00299 BC00299 V=1000.0  +MOVJ EC00299
SFTOF3D
MOVJ C00300 BC00300 VJ=100.00  +MOVJ EC00300 VJ=100.00
'Path W383
SFTOF3D
SFTON3D P046
MOVJ C00301 BC00301 VJ=100.00  +MOVJ EC00301 VJ=100.00
MOVJ C00302 BC00302 VJ=100.00  +MOVJ EC00302 VJ=100.00
SMOVL C00303 BC00303 V=400.0  +MOVJ EC00303
SMOVL C00304 BC00304 V=133.3 PL=0  +MOVJ EC00304
SREFP 1 C00305 BC00305  +REFP EC00305
SREFP 2 C00306 BC00306  +REFP EC00306
ARCON
SMOVL C00307 BC00307 V=9.2  +MOVJ EC00307
SMOVL C00308 BC00308 V=9.2  +MOVJ EC00308
SMOVL C00309 BC00309 V=9.2  +MOVJ EC00309
ARCOF
SMOVL C00310 BC00310 V=400.0  +MOVJ EC00310
SMOVL C00311 BC00311 V=1000.0  +MOVJ EC00311
SFTOF3D
MOVJ C00312 BC00312 VJ=100.00  +MOVJ EC00312 VJ=100.00
MOVJ C00313 BC00313 VJ=100.00  +MOVJ EC00313 VJ=100.00
'Down
MOVJ C00314 BC00314 VJ=100.00  +MOVJ EC00314 VJ=100.00
MOVJ C00315 BC00315 VJ=100.00  +MOVJ EC00315 VJ=100.00
'Path W1720
SFTOF3D
SFTON3D P032
MOVJ C00316 BC00316 VJ=100.00  +MOVJ EC00316 VJ=100.00
SMOVL C00317 BC00317 V=400.0  +MOVJ EC00317
SMOVL C00318 BC00318 V=133.3  +MOVJ EC00318
SREFP 1 C00319 BC00319  +REFP EC00319
SREFP 2 C00320 BC00320  +REFP EC00320
MACRO1 MJ#(0) ARGF21
ARCON
SWVON WEV#(100)
SMOVC C00321 BC00321 V=9.2  +MOVJ EC00321
SMOVC C00322 BC00322 V=9.2  +MOVJ EC00322
SMOVC C00323 BC00323 V=9.2  +MOVJ EC00323
SMOVC C00324 BC00324 V=9.2  +MOVJ EC00324
SMOVC C00325 BC00325 V=9.2  +MOVJ EC00325
SMOVC C00326 BC00326 V=9.2  +MOVJ EC00326
ARCOF
SWVOF
SMOVL C00327 BC00327 V=400.0  +MOVJ EC00327
SMOVL C00328 BC00328 V=1000.0  +MOVJ EC00328
SFTOF3D
MOVJ C00329 BC00329 VJ=100.00  +MOVJ EC00329 VJ=100.00
MOVJ C00330 BC00330 VJ=100.00  +MOVJ EC00330 VJ=100.00
MOVJ C00331 BC00331 VJ=100.00  +MOVJ EC00331 VJ=100.00
MOVJ C00332 BC00332 VJ=100.00  +MOVJ EC00332 VJ=100.00
MOVJ C00333 BC00333 VJ=100.00  +MOVJ EC00333 VJ=100.00
MOVJ C00334 BC00334 VJ=100.00  +MOVJ EC00334 VJ=100.00
'Path W1626
SFTOF3D
COMM SFTON3D P022
COMM MOVJ C00335 BC00335 VJ=100.00  +MOVJ EC00335 VJ=100.00
COMM SMOVL C00336 BC00336 V=250.0  +MOVJ EC00336
COMM SMOVL C00337 BC00337 V=133.3 PL=0  +MOVJ EC00337
COMM SREFP 1 C00338 BC00338  +REFP EC00338
COMM SREFP 2 C00339 BC00339  +REFP EC00339
COMM MACRO1 MJ#(0) ARGF9
COMM ARCON
COMM SMOVC C00340 BC00340 V=9.2  +MOVJ EC00340
COMM SMOVC C00341 BC00341 V=10.0  +MOVJ EC00341
COMM SMOVC C00342 BC00342 V=10.0  +MOVJ EC00342
COMM SMOVC C00343 BC00343 V=10.0  +MOVJ EC00343
COMM SMOVC C00344 BC00344 V=10.0  +MOVJ EC00344
COMM SMOVC C00345 BC00345 V=10.0  +MOVJ EC00345
COMM SMOVC C00346 BC00346 V=10.0  +MOVJ EC00346
COMM ARCOF
COMM SMOVL C00347 BC00347 V=400.0  +MOVJ EC00347
COMM SMOVL C00348 BC00348 V=400.0  +MOVJ EC00348
COMM SFTOF3D
COMM 'Path W1627
COMM SFTOF3D
COMM SFTON3D P022
COMM MOVJ C00349 BC00349 VJ=20.00  +MOVJ EC00349 VJ=100.00
COMM SMOVL C00350 BC00350 V=133.3  +MOVJ EC00350
COMM SMOVL C00351 BC00351 V=100.0 PL=0  +MOVJ EC00351
COMM SREFP 1 C00352 BC00352  +REFP EC00352
COMM SREFP 2 C00353 BC00353  +REFP EC00353
COMM ARCON
COMM SMOVL C00354 BC00354 V=10.0  +MOVJ EC00354
COMM SMOVL C00355 BC00355 V=10.0  +MOVJ EC00355
COMM SMOVL C00356 BC00356 V=13.3  +MOVJ EC00356
COMM ARCOF
COMM SMOVL C00357 BC00357 V=400.0  +MOVJ EC00357
COMM SMOVL C00358 BC00358 V=1000.0  +MOVJ EC00358
SFTOF3D
MOVJ C00359 BC00359 VJ=100.00  +MOVJ EC00359 VJ=100.00
MOVJ C00360 BC00360 VJ=100.00  +MOVJ EC00360 VJ=100.00
MACRO1 MJ#(0) ARGF14
SFTON3D P066
SMOVL C00361 BC00361 V=166.7  +MOVJ EC00361
ARCON
SMOVL C00362 BC00362 V=11.7  +MOVJ EC00362
ARCOF
SMOVL C00363 BC00363 V=333.3  +MOVJ EC00363
SFTOF3D
MOVJ C00364 BC00364 VJ=100.00  +MOVJ EC00364 VJ=100.00
MOVJ C00365 BC00365 VJ=100.00  +MOVJ EC00365 VJ=100.00
SMOVL C00366 BC00366 V=666.7  +MOVJ EC00366
SFTON3D P068
SMOVL C00367 BC00367 V=166.7  +MOVJ EC00367
ARCON
SMOVL C00368 BC00368 V=12.5  +MOVJ EC00368
SMOVL C00369 BC00369 V=10.8  +MOVJ EC00369
SMOVL C00370 BC00370 V=10.8  +MOVJ EC00370
ARCOF
SMOVL C00371 BC00371 V=166.7  +MOVJ EC00371
SMOVL C00372 BC00372 V=666.7  +MOVJ EC00372
SFTOF3D
SMOVL C00373 BC00373 V=666.7  +MOVJ EC00373
'
MOVJ C00374 BC00374 VJ=100.00  +MOVJ EC00374 VJ=100.00
MOVJ C00375 BC00375 VJ=100.00  +MOVJ EC00375 VJ=100.00
MOVJ C00376 BC00376 VJ=100.00  +MOVJ EC00376 VJ=100.00
'Path W1911
SFTOF3D
MOVJ C00377 BC00377 VJ=100.00  +MOVJ EC00377 VJ=100.00
SMOVL C00378 BC00378 V=166.7  +MOVJ EC00378
SFTON3D P021
SMOVL C00379 BC00379 V=100.0 PL=0  +MOVJ EC00379
SREFP 1 C00380 BC00380  +REFP EC00380
SREFP 2 C00381 BC00381  +REFP EC00381
MACRO1 MJ#(0) ARGF21
ARCON
SWVON WEV#(100)
SMOVC C00382 BC00382 V=9.2  +MOVJ EC00382
SMOVC C00383 BC00383 V=9.2  +MOVJ EC00383
SMOVC C00384 BC00384 V=9.2  +MOVJ EC00384
SMOVC C00385 BC00385 V=9.2  +MOVJ EC00385
ARCOF
SWVOF
SMOVL C00386 BC00386 V=400.0  +MOVJ EC00386
SMOVL C00387 BC00387 V=1000.0  +MOVJ EC00387
SFTOF3D
MOVJ C00388 BC00388 VJ=100.00  +MOVJ EC00388 VJ=100.00
'
MOVJ C00389 BC00389 VJ=100.00  +MOVJ EC00389 VJ=100.00
MOVJ C00390 BC00390 VJ=100.00  +MOVJ EC00390 VJ=100.00
'NIE SPAWAMY
COMM 'Path W1642
COMM SFTOF3D
COMM SFTON3D P024
COMM MOVJ C00391 BC00391 VJ=100.00  +MOVJ EC00391 VJ=100.00
COMM SMOVL C00392 BC00392 V=400.0  +MOVJ EC00392
COMM SMOVL C00393 BC00393 V=100.0 PL=0  +MOVJ EC00393
COMM SREFP 1 C00394 BC00394  +REFP EC00394
COMM SREFP 2 C00395 BC00395  +REFP EC00395
COMM MACRO1 MJ#(0) ARGF0
COMM ARCON
COMM SMOVL C00396 BC00396 V=10.0  +MOVJ EC00396
COMM ARCOF
COMM SMOVL C00397 BC00397 V=400.0  +MOVJ EC00397
COMM SMOVL C00398 BC00398 V=1000.0  +MOVJ EC00398
COMM SFTOF3D
'NIE SPAWAMY
COMM 'Path W1643
COMM SFTOF3D
COMM SFTON3D P025
COMM MOVJ C00399 BC00399 VJ=100.00  +MOVJ EC00399 VJ=100.00
COMM SMOVL C00400 BC00400 V=400.0  +MOVJ EC00400
COMM SMOVL C00401 BC00401 V=100.0 PL=0  +MOVJ EC00401
COMM SREFP 1 C00402 BC00402  +REFP EC00402
COMM SREFP 2 C00403 BC00403  +REFP EC00403
COMM MACRO1 MJ#(0) ARGF0
COMM ARCON
COMM SMOVL C00404 BC00404 V=10.0  +MOVJ EC00404
COMM ARCOF
COMM SMOVL C00405 BC00405 V=400.0  +MOVJ EC00405
COMM SMOVL C00406 BC00406 V=1000.0  +MOVJ EC00406
COMM SMOVL C00407 BC00407 V=1000.0  +MOVJ EC00407
COMM SFTOF3D
'
'Path W1644
SFTOF3D
SFTON3D P026
MOVJ C00408 BC00408 VJ=100.00  +MOVJ EC00408 VJ=100.00
SMOVL C00409 BC00409 V=333.3  +MOVJ EC00409
SMOVL C00410 BC00410 V=133.3 PL=0  +MOVJ EC00410
SREFP 1 C00411 BC00411  +REFP EC00411
SREFP 2 C00412 BC00412  +REFP EC00412
MACRO1 MJ#(0) ARGF9
ARCON
SMOVL C00413 BC00413 V=6.7  +MOVJ EC00413
SMOVL C00414 BC00414 V=6.7  +MOVJ EC00414
SMOVL C00415 BC00415 V=6.7  +MOVJ EC00415
SMOVL C00416 BC00416 V=5.0  +MOVJ EC00416
SMOVL C00417 BC00417 V=5.0  +MOVJ EC00417
SMOVL C00418 BC00418 V=5.0  +MOVJ EC00418
ARCOF
SMOVL C00419 BC00419 V=133.3  +MOVJ EC00419
SMOVL C00420 BC00420 V=333.3  +MOVJ EC00420
SMOVL C00421 BC00421 V=333.3  +MOVJ EC00421
SFTOF3D
'Path W1645
SFTOF3D
SFTON3D P027
MOVJ C00422 BC00422 VJ=50.00  +MOVJ EC00422 VJ=100.00
SMOVL C00423 BC00423 V=166.7  +MOVJ EC00423
SMOVL C00424 BC00424 V=133.3 PL=0  +MOVJ EC00424
SREFP 1 C00425 BC00425  +REFP EC00425
SREFP 2 C00426 BC00426  +REFP EC00426
MACRO1 MJ#(0) ARGF9
ARCON
SMOVL C00427 BC00427 V=6.7  +MOVJ EC00427
SMOVL C00428 BC00428 V=6.7  +MOVJ EC00428
SMOVL C00429 BC00429 V=6.7  +MOVJ EC00429
ARCON
SMOVL C00430 BC00430 V=6.7  +MOVJ EC00430
SMOVL C00431 BC00431 V=6.7  +MOVJ EC00431
ARCOF
SMOVL C00432 BC00432 V=400.0  +MOVJ EC00432
SMOVL C00433 BC00433 V=1000.0  +MOVJ EC00433
SMOVL C00434 BC00434 V=1000.0  +MOVJ EC00434
SFTOF3D
MOVJ C00435 BC00435 VJ=40.00  +MOVJ EC00435 VJ=100.00
MOVJ C00436 BC00436 VJ=100.00  +MOVJ EC00436 VJ=100.00
MOVL C00437 BC00437 V=1000.0  +MOVJ EC00437 VJ=100.00
MOVL C00438 BC00438 V=1000.0  +MOVJ EC00438 VJ=100.00
MOVL C00439 BC00439 V=1000.0  +MOVJ EC00439 VJ=100.00
MOVL C00440 BC00440 V=1000.0  +MOVJ EC00440 VJ=100.00
SFTON3D P051
SMOVL C00441 BC00441 V=166.7 PL=0  +MOVJ EC00441
ARCON
SMOVL C00442 BC00442 V=13.3  +MOVJ EC00442
SMOVC C00443 BC00443 V=15.0  +MOVJ EC00443
SMOVC C00444 BC00444 V=15.0  +MOVJ EC00444
SMOVC C00445 BC00445 V=15.0  +MOVJ EC00445
SMOVL C00446 BC00446 V=6.7  +MOVJ EC00446
SFTON3D P052
SMOVL C00447 BC00447 V=11.7  +MOVJ EC00447
ARCOF
SMOVL C00448 BC00448 V=166.7  +MOVJ EC00448
SFTOF3D
SMOVL C00449 BC00449 V=666.7  +MOVJ EC00449
SFTON3D P054
SMOVL C00450 BC00450 V=166.7 PL=0  +MOVJ EC00450
ARCON
SMOVL C00451 BC00451 V=13.3  +MOVJ EC00451
SMOVL C00452 BC00452 V=15.0  +MOVJ EC00452
SMOVL C00453 BC00453 V=15.0  +MOVJ EC00453
SMOVL C00454 BC00454 V=15.0  +MOVJ EC00454
SMOVL C00455 BC00455 V=12.5  +MOVJ EC00455
SFTON3D P053
SMOVL C00456 BC00456 V=12.5  +MOVJ EC00456
ARCOF
SMOVL C00457 BC00457 V=166.7  +MOVJ EC00457
SFTOF3D
SMOVL C00458 BC00458 V=666.7  +MOVJ EC00458
SFTON3D P055
SMOVL C00459 BC00459 V=166.7 PL=0  +MOVJ EC00459
ARCON
SMOVL C00460 BC00460 V=15.0  +MOVJ EC00460
SMOVL C00461 BC00461 V=15.0  +MOVJ EC00461
SMOVL C00462 BC00462 V=15.0  +MOVJ EC00462
SMOVL C00463 BC00463 V=12.5  +MOVJ EC00463
SFTON3D P056
SMOVL C00464 BC00464 V=12.5  +MOVJ EC00464
SMOVL C00465 BC00465 V=15.0  +MOVJ EC00465
SMOVL C00466 BC00466 V=15.0  +MOVJ EC00466
ARCOF
SMOVL C00467 BC00467 V=166.7  +MOVJ EC00467
SFTOF3D
SMOVL C00468 BC00468 V=666.7  +MOVJ EC00468
SMOVL C00469 BC00469 V=666.7  +MOVJ EC00469
COMM 'jakie searche do takicj spoin?
COMM MOVJ C00470 BC00470 VJ=100.00  +MOVJ EC00470 VJ=100.00
COMM 'Path W1646
COMM SFTOF3D
COMM MOVJ C00471 BC00471 VJ=100.00  +MOVJ EC00471 VJ=100.00
COMM MOVL C00472 BC00472 V=400.0  +MOVJ EC00472 VJ=100.00
COMM PAUSE
COMM PAUSE
'USUNAC SPAWANIE ZAMKOW
COMM SFTOF3D
COMM SFTON3D P021
COMM SMOVL C00473 BC00473 V=166.7 PL=0  +MOVJ EC00473
COMM SREFP 1 C00474 BC00474  +REFP EC00474
COMM SREFP 2 C00475 BC00475  +REFP EC00475
COMM MACRO1 MJ#(0) ARGF6
COMM ARCON
COMM SMOVL C00476 BC00476 V=4.2  +MOVJ EC00476
COMM ARCOF
COMM MOVL C00477 BC00477 V=400.0  +MOVJ EC00477 VJ=100.00
COMM MOVL C00478 BC00478 V=1000.0  +MOVJ EC00478 VJ=100.00
COMM MOVL C00479 BC00479 V=333.3  +MOVJ EC00479 VJ=100.00
COMM MOVJ C00480 BC00480 VJ=100.00  +MOVJ EC00480 VJ=100.00
COMM 'brak dostÃÂpu do jednej spoiny
COMM 'Path W1647
COMM SFTOF3D
COMM MOVJ C00481 BC00481 VJ=25.00  +MOVJ EC00481 VJ=100.00
COMM MOVJ C00482 BC00482 VJ=25.00  +MOVJ EC00482 VJ=100.00
COMM MOVL C00483 BC00483 V=400.0  +MOVJ EC00483 VJ=100.00
COMM SFTOF3D
COMM SMOVL C00484 BC00484 V=166.7 PL=0  +MOVJ EC00484
COMM SREFP 1 C00485 BC00485  +REFP EC00485
COMM SREFP 2 C00486 BC00486  +REFP EC00486
COMM MACRO1 MJ#(0) ARGF6
COMM ARCON
COMM SMOVL C00487 BC00487 V=4.2  +MOVJ EC00487
COMM ARCOF
COMM MOVL C00488 BC00488 V=400.0  +MOVJ EC00488 VJ=100.00
COMM MOVL C00489 BC00489 V=1000.0  +MOVJ EC00489 VJ=100.00
COMM 'Path W1648
COMM SFTOF3D
COMM MOVJ C00490 BC00490 VJ=10.00  +MOVJ EC00490 VJ=100.00
COMM MOVL C00491 BC00491 V=166.7  +MOVJ EC00491 VJ=100.00
COMM SFTON3D P021
COMM SMOVL C00492 BC00492 V=100.0 PL=0  +MOVJ EC00492
COMM SREFP 1 C00493 BC00493  +REFP EC00493
COMM SREFP 2 C00494 BC00494  +REFP EC00494
COMM MACRO1 MJ#(0) ARGF6
COMM ARCON
COMM SMOVL C00495 BC00495 V=4.2  +MOVJ EC00495
COMM ARCOF
COMM MOVL C00496 BC00496 V=400.0  +MOVJ EC00496 VJ=100.00
COMM MOVL C00497 BC00497 V=1000.0  +MOVJ EC00497 VJ=100.00
COMM MOVL C00498 BC00498 V=1000.0  +MOVJ EC00498 VJ=100.00
COMM MOVJ C00499 BC00499 VJ=10.00  +MOVJ EC00499 VJ=100.00
COMM 'Path W1649
COMM SFTOF3D
COMM MOVJ C00500 BC00500 VJ=15.00  +MOVJ EC00500 VJ=100.00
COMM MOVL C00501 BC00501 V=166.7  +MOVJ EC00501 VJ=100.00
COMM SFTON3D P021
COMM SMOVL C00502 BC00502 V=166.7 PL=0  +MOVJ EC00502
COMM SREFP 1 C00503 BC00503  +REFP EC00503
COMM SREFP 2 C00504 BC00504  +REFP EC00504
COMM MACRO1 MJ#(0) ARGF6
COMM ARCON
COMM SMOVL C00505 BC00505 V=4.2  +MOVJ EC00505
COMM ARCOF
COMM MOVL C00506 BC00506 V=400.0  +MOVJ EC00506 VJ=100.00
COMM MOVL C00507 BC00507 V=1000.0  +MOVJ EC00507 VJ=100.00
COMM 'Path W1650
COMM MOVJ C00508 BC00508 VJ=100.00  +MOVJ EC00508 VJ=100.00
COMM MOVL C00509 BC00509 V=166.7  +MOVJ EC00509 VJ=100.00
COMM SMOVL C00510 BC00510 V=166.7 PL=0  +MOVJ EC00510
COMM SREFP 1 C00511 BC00511  +REFP EC00511
COMM SREFP 2 C00512 BC00512  +REFP EC00512
COMM MACRO1 MJ#(0) ARGF6
COMM ARCON
COMM SMOVL C00513 BC00513 V=4.2  +MOVJ EC00513
COMM ARCOF
COMM MOVL C00514 BC00514 V=400.0  +MOVJ EC00514 VJ=100.00
COMM MOVL C00515 BC00515 V=1000.0  +MOVJ EC00515 VJ=100.00
COMM 'Path W1651
COMM SFTOF3D
COMM MOVJ C00516 BC00516 VJ=100.00  +MOVJ EC00516 VJ=100.00
COMM MOVL C00517 BC00517 V=400.0  +MOVJ EC00517 VJ=100.00
COMM SFTON3D P021
COMM SMOVL C00518 BC00518 V=166.7 PL=0  +MOVJ EC00518
COMM SREFP 1 C00519 BC00519  +REFP EC00519
COMM SREFP 2 C00520 BC00520  +REFP EC00520
COMM MACRO1 MJ#(0) ARGF6
COMM ARCON
COMM SMOVL C00521 BC00521 V=4.2  +MOVJ EC00521
COMM ARCOF
COMM MOVL C00522 BC00522 V=400.0  +MOVJ EC00522 VJ=100.00
COMM MOVL C00523 BC00523 V=1000.0  +MOVJ EC00523 VJ=100.00
COMM 'Path W1652
COMM SFTOF3D
COMM MOVJ C00524 BC00524 VJ=100.00  +MOVJ EC00524 VJ=100.00
COMM MOVL C00525 BC00525 V=166.7  +MOVJ EC00525 VJ=100.00
COMM SFTON3D P021
COMM SMOVL C00526 BC00526 V=166.7 PL=0  +MOVJ EC00526
COMM SREFP 1 C00527 BC00527  +REFP EC00527
COMM SREFP 2 C00528 BC00528  +REFP EC00528
COMM MACRO1 MJ#(0) ARGF6
COMM ARCON
COMM SMOVL C00529 BC00529 V=4.2  +MOVJ EC00529
COMM ARCOF
COMM MOVL C00530 BC00530 V=166.7  +MOVJ EC00530 VJ=100.00
COMM MOVL C00531 BC00531 V=166.7  +MOVJ EC00531 VJ=100.00
COMM MOVJ C00532 BC00532 VJ=50.00  +MOVJ EC00532 VJ=20.00
COMM SMOVL C00533 BC00533 V=166.7  +MOVJ EC00533
COMM ARCON
COMM SMOVL C00534 BC00534 V=4.2  +MOVJ EC00534
COMM ARCOF
COMM SMOVL C00535 BC00535 V=166.7  +MOVJ EC00535
COMM 'jakie searche do takicj spoin?
COMM MOVJ C00536 BC00536 VJ=100.00  +MOVJ EC00536 VJ=100.00
COMM MOVJ C00537 BC00537 VJ=20.00  +MOVJ EC00537 VJ=100.00
COMM MOVJ C00538 BC00538 VJ=100.00  +MOVJ EC00538 VJ=100.00
COMM MOVJ C00539 BC00539 VJ=100.00  +MOVJ EC00539 VJ=100.00
COMM 'Path W1653
COMM SFTOF3D
COMM MOVJ C00540 BC00540 VJ=100.00  +MOVJ EC00540 VJ=100.00
COMM MOVL C00541 BC00541 V=166.7  +MOVJ EC00541 VJ=100.00
COMM SFTON3D P067
COMM SMOVL C00542 BC00542 V=166.7 PL=0  +MOVJ EC00542
COMM SREFP 1 C00543 BC00543  +REFP EC00543
COMM SREFP 2 C00544 BC00544  +REFP EC00544
COMM ARCON
COMM MACRO1 MJ#(0) ARGF9
COMM SMOVL C00545 BC00545 V=10.8  +MOVJ EC00545
COMM ARCOF
COMM SMOVL C00546 BC00546 V=166.7  +MOVJ EC00546
COMM SMOVL C00547 BC00547 V=666.7  +MOVJ EC00547
COMM SMOVL C00548 BC00548 V=166.7  +MOVJ EC00548
COMM ARCON
COMM SMOVL C00549 BC00549 V=10.8  +MOVJ EC00549
COMM ARCOF
COMM SMOVL C00550 BC00550 V=250.0  +MOVJ EC00550
COMM 'Path W1654
COMM SFTOF3D
COMM MOVJ C00551 BC00551 VJ=100.00  +MOVJ EC00551 VJ=100.00
COMM MOVJ C00552 BC00552 VJ=100.00  +MOVJ EC00552 VJ=100.00
MOVJ C00553 BC00553 VJ=100.00  +MOVJ EC00553 VJ=100.00
'Down
END
